C07321=1192.397,329.758,-73.014,-176.371,7.845,148.458
C07322=1192.393,330.005,-73.045,-176.368,7.848,148.458
C07323=1192.389,330.253,-73.077,-176.366,7.851,148.458
C07324=1192.384,330.501,-73.109,-176.363,7.855,148.459
C07325=1192.381,330.749,-73.141,-176.361,7.858,148.459
C07326=1192.377,330.997,-73.173,-176.359,7.860,148.459
C07327=1192.372,331.245,-73.205,-176.357,7.864,148.459
C07328=1192.368,331.493,-73.237,-176.354,7.867,148.459
C07329=1192.364,331.741,-73.268,-176.352,7.870,148.459
C07330=1192.359,331.989,-73.300,-176.350,7.873,148.459
C07331=1192.355,332.237,-73.332,-176.347,7.875,148.459
C07332=1192.352,332.485,-73.363,-176.345,7.879,148.460
C07333=1192.347,332.733,-73.395,-176.342,7.882,148.460
C07334=1192.343,332.981,-73.427,-176.340,7.885,148.460
C07335=1192.339,333.229,-73.459,-176.338,7.888,148.460
C07336=1192.334,333.476,-73.491,-176.335,7.892,148.460
C07337=1192.331,333.724,-73.524,-176.334,7.894,148.460
C07338=1192.327,333.972,-73.556,-176.331,7.897,148.460
C07339=1192.322,334.220,-73.588,-176.329,7.900,148.460
C07340=1192.318,334.468,-73.620,-176.326,7.904,148.461
C07341=1192.314,334.716,-73.652,-176.324,7.907,148.461
C07342=1192.310,334.963,-73.683,-176.321,7.910,148.461
C07343=1192.305,335.212,-73.716,-176.320,7.913,148.461
C07344=1192.301,335.460,-73.748,-176.318,7.916,148.461
C07345=1192.298,335.708,-73.780,-176.315,7.919,148.461
C07346=1192.293,335.955,-73.812,-176.313,7.922,148.461
C07347=1192.289,336.203,-73.844,-176.310,7.926,148.462
C07348=1192.285,336.451,-73.877,-176.308,7.929,148.462
C07349=1192.281,336.699,-73.909,-176.306,7.931,148.462
C07350=1192.276,336.947,-73.941,-176.304,7.934,148.462
C07351=1192.273,337.194,-73.973,-176.302,7.938,148.462
C07352=1192.268,337.443,-74.006,-176.299,7.941,148.462
C07353=1192.265,337.691,-74.037,-176.297,7.944,148.463
C07354=1192.260,337.938,-74.070,-176.294,7.947,148.463
C07355=1192.256,338.186,-74.102,-176.293,7.950,148.463
C07356=1192.252,338.434,-74.135,-176.290,7.953,148.463
C07357=1192.248,338.682,-74.166,-176.288,7.956,148.463
C07358=1192.244,338.930,-74.199,-176.286,7.960,148.463
C07359=1192.240,339.177,-74.231,-176.283,7.963,148.464
C07360=1192.235,339.425,-74.263,-176.281,7.966,148.464
C07361=1192.231,339.674,-74.296,-176.279,7.969,148.464
C07362=1192.227,339.921,-74.328,-176.277,7.972,148.464
C07363=1192.223,340.200,-74.365,-176.274,7.976,148.464
C07364=1192.218,340.479,-74.401,-176.272,7.979,148.464
C07365=1192.212,340.757,-74.438,-176.269,7.982,148.465
C07366=1192.208,341.036,-74.474,-176.267,7.987,148.465
C07367=1192.204,341.284,-74.506,-176.265,7.989,148.465
C07368=1192.200,341.531,-74.539,-176.263,7.992,148.465
C07369=1192.195,341.780,-74.572,-176.260,7.996,148.465
C07370=1192.192,342.027,-74.604,-176.258,7.999,148.466
C07371=1192.188,342.276,-74.637,-176.255,8.002,148.466
C07372=1192.183,342.523,-74.669,-176.253,8.005,148.466
C07373=1192.179,342.771,-74.701,-176.252,8.008,148.466
C07374=1192.175,343.018,-74.734,-176.249,8.011,148.466
C07375=1192.171,343.267,-74.767,-176.247,8.015,148.467
C07376=1192.167,343.514,-74.799,-176.245,8.018,148.467
C07377=1192.163,343.763,-74.832,-176.243,8.021,148.467
C07378=1192.159,344.010,-74.865,-176.240,8.025,148.467
C07379=1192.154,344.257,-74.898,-176.239,8.027,148.467
C07380=1192.150,344.505,-74.930,-176.236,8.030,148.468
C07381=1192.146,344.753,-74.963,-176.234,8.034,148.468
C07382=1192.142,345.001,-74.995,-176.232,8.037,148.468
C07383=1192.137,345.249,-75.028,-176.230,8.040,148.468
C07384=1192.134,345.497,-75.061,-176.227,8.044,148.468
C07385=1192.130,345.745,-75.093,-176.226,8.046,148.469
C07386=1192.125,345.993,-75.127,-176.224,8.050,148.469
C07387=1192.121,346.240,-75.160,-176.221,8.053,148.469
C07388=1192.118,346.488,-75.192,-176.219,8.056,148.469
C07389=1192.113,346.736,-75.225,-176.217,8.060,148.470
C07390=1192.109,346.983,-75.258,-176.215,8.063,148.470
C07391=1192.104,347.231,-75.290,-176.213,8.065,148.470
C07392=1192.100,347.479,-75.323,-176.211,8.069,148.470
C07393=1192.096,347.727,-75.356,-176.208,8.072,148.470
C07394=1192.093,347.974,-75.389,-176.206,8.075,148.471
C07395=1192.088,348.223,-75.421,-176.204,8.079,148.471
C07396=1192.084,348.470,-75.454,-176.202,8.082,148.471
C07397=1192.080,348.718,-75.488,-176.199,8.085,148.471
C07398=1192.076,348.966,-75.521,-176.198,8.088,148.471
C07399=1192.072,349.214,-75.554,-176.196,8.091,148.472
C07400=1192.067,349.461,-75.587,-176.194,8.095,148.472
C07401=1192.063,349.710,-75.620,-176.191,8.098,148.472
C07402=1192.060,349.957,-75.652,-176.189,8.101,148.473
C07403=1192.056,350.205,-75.685,-176.187,8.105,148.473
C07404=1192.051,350.453,-75.718,-176.185,8.107,148.473
C07405=1192.047,350.700,-75.752,-176.183,8.111,148.473
C07406=1192.043,350.948,-75.785,-176.181,8.114,148.474
C07407=1192.039,351.196,-75.818,-176.179,8.118,148.474
C07408=1192.035,351.444,-75.851,-176.177,8.121,148.474
C07409=1192.031,351.691,-75.884,-176.175,8.124,148.474
C07410=1192.027,351.939,-75.917,-176.173,8.127,148.474
C07411=1192.022,352.187,-75.951,-176.171,8.130,148.475
C07412=1192.018,352.434,-75.984,-176.169,8.134,148.475
C07413=1192.014,352.682,-76.017,-176.167,8.137,148.475
C07414=1192.010,352.930,-76.050,-176.164,8.140,148.476
C07415=1192.006,353.178,-76.083,-176.163,8.144,148.476
C07416=1192.002,353.425,-76.116,-176.161,8.146,148.476
C07417=1191.998,353.674,-76.150,-176.159,8.150,148.476
C07418=1191.994,353.922,-76.183,-176.156,8.153,148.477
C07419=1191.990,354.169,-76.216,-176.155,8.157,148.477
C07420=1191.986,354.417,-76.249,-176.152,8.160,148.477
C07421=1191.982,354.665,-76.282,-176.150,8.163,148.477
C07422=1191.977,354.912,-76.316,-176.149,8.166,148.478
C07423=1191.973,355.160,-76.349,-176.147,8.169,148.478
C07424=1191.969,355.408,-76.382,-176.144,8.173,148.478
C07425=1191.965,355.656,-76.415,-176.143,8.176,148.479
C07426=1191.961,355.903,-76.449,-176.140,8.180,148.479
C07427=1191.957,356.150,-76.482,-176.139,8.183,148.479
C07428=1191.953,356.399,-76.516,-176.137,8.186,148.480
C07429=1191.949,356.647,-76.549,-176.135,8.189,148.480
C07430=1191.945,356.895,-76.583,-176.133,8.193,148.480
C07431=1191.941,357.142,-76.616,-176.131,8.196,148.480
C07432=1191.937,357.389,-76.650,-176.129,8.200,148.481
C07433=1191.932,357.637,-76.683,-176.127,8.203,148.481
C07434=1191.928,357.885,-76.716,-176.125,8.206,148.481
C07435=1191.925,358.133,-76.750,-176.123,8.209,148.482
C07436=1191.920,358.381,-76.784,-176.121,8.213,148.482
C07437=1191.916,358.629,-76.817,-176.119,8.216,148.482
C07438=1191.912,358.876,-76.850,-176.117,8.220,148.483
C07439=1191.908,359.123,-76.884,-176.115,8.223,148.483
C07440=1191.904,359.371,-76.917,-176.113,8.226,148.483
C07441=1191.900,359.620,-76.951,-176.112,8.229,148.484
C07442=1191.896,359.867,-76.985,-176.110,8.233,148.484
C07443=1191.892,360.115,-77.018,-176.108,8.236,148.484
C07444=1191.888,360.362,-77.052,-176.106,8.240,148.485
C07445=1191.884,360.610,-77.085,-176.104,8.242,148.485
C07446=1191.879,360.858,-77.119,-176.102,8.246,148.485
C07447=1191.876,361.105,-77.153,-176.100,8.249,148.486
C07448=1191.871,361.353,-77.186,-176.098,8.253,148.486
C07449=1191.868,361.600,-77.220,-176.097,8.256,148.486
C07450=1191.863,361.848,-77.254,-176.095,8.259,148.487
C07451=1191.860,362.096,-77.288,-176.093,8.263,148.487
C07452=1191.855,362.344,-77.322,-176.091,8.266,148.488
C07453=1191.851,362.592,-77.355,-176.090,8.269,148.488
C07454=1191.847,362.839,-77.389,-176.088,8.273,148.488
C07455=1191.843,363.087,-77.423,-176.086,8.276,148.489
C07456=1191.839,363.334,-77.457,-176.084,8.280,148.489
C07457=1191.836,363.582,-77.490,-176.082,8.282,148.489
C07458=1191.831,363.830,-77.524,-176.081,8.286,148.490
C07459=1191.827,364.077,-77.558,-176.079,8.290,148.490
C07460=1191.823,364.325,-77.592,-176.078,8.292,148.490
C07461=1191.819,364.573,-77.626,-176.076,8.296,148.491
C07462=1191.815,364.820,-77.659,-176.074,8.299,148.491
C07463=1191.811,365.068,-77.693,-176.072,8.302,148.491
C07464=1191.807,365.316,-77.728,-176.071,8.306,148.492
C07465=1191.803,365.563,-77.761,-176.069,8.309,148.492
C07466=1191.799,365.811,-77.796,-176.068,8.312,148.493
C07467=1191.794,366.092,-77.834,-176.065,8.317,148.493
C07468=1191.789,366.373,-77.872,-176.063,8.320,148.494
C07469=1191.785,366.655,-77.911,-176.062,8.324,148.494
C07470=1191.780,366.935,-77.949,-176.060,8.328,148.495
C07471=1191.777,367.183,-77.984,-176.058,8.331,148.495
C07472=1191.772,367.431,-78.017,-176.057,8.334,148.495
C07473=1191.768,367.678,-78.051,-176.055,8.338,148.496
C07474=1191.764,367.926,-78.086,-176.054,8.340,148.496
C07475=1191.760,368.174,-78.119,-176.052,8.344,148.497
C07476=1191.756,368.421,-78.153,-176.050,8.348,148.497
C07477=1191.752,368.669,-78.188,-176.049,8.350,148.497
C07478=1191.748,368.916,-78.222,-176.047,8.354,148.498
C07479=1191.744,369.164,-78.256,-176.046,8.357,148.498
C07480=1191.740,369.412,-78.290,-176.044,8.360,148.499
C07481=1191.736,369.660,-78.324,-176.043,8.363,148.499
C07482=1191.732,369.907,-78.358,-176.041,8.367,148.500
C07483=1191.728,370.155,-78.393,-176.040,8.371,148.500
C07484=1191.724,370.402,-78.427,-176.039,8.374,148.501
C07485=1191.719,370.650,-78.461,-176.037,8.377,148.501
C07486=1191.716,370.898,-78.495,-176.035,8.380,148.501
C07487=1191.711,371.145,-78.529,-176.034,8.384,148.502
C07488=1191.707,371.392,-78.563,-176.032,8.386,148.502
C07489=1191.704,371.640,-78.598,-176.031,8.390,148.503
C07490=1191.700,371.888,-78.632,-176.030,8.393,148.503
C07491=1191.696,372.136,-78.667,-176.029,8.396,148.504
C07492=1191.692,372.383,-78.701,-176.027,8.400,148.504
C07493=1191.687,372.631,-78.734,-176.026,8.403,148.505
C07494=1191.683,372.879,-78.769,-176.024,8.406,148.505
C07495=1191.679,373.126,-78.803,-176.023,8.409,148.505
C07496=1191.675,373.374,-78.838,-176.021,8.413,148.506
C07497=1191.671,373.621,-78.872,-176.020,8.416,148.506
C07498=1191.667,373.869,-78.906,-176.019,8.420,148.507
C07499=1191.663,374.117,-78.941,-176.017,8.422,148.507
C07500=1191.659,374.364,-78.975,-176.017,8.425,148.508
C07501=1191.655,374.612,-79.010,-176.015,8.429,148.508
C07502=1191.651,374.859,-79.044,-176.014,8.432,148.509
C07503=1191.647,375.107,-79.078,-176.013,8.435,148.509
C07504=1191.643,375.355,-79.113,-176.011,8.439,148.510
C07505=1191.639,375.602,-79.147,-176.010,8.442,148.510
C07506=1191.635,375.850,-79.182,-176.009,8.444,148.511
C07507=1191.631,376.097,-79.216,-176.008,8.448,148.511
C07508=1191.627,376.345,-79.250,-176.006,8.451,148.512
C07509=1191.623,376.592,-79.286,-176.006,8.454,148.512
C07510=1191.620,376.840,-79.320,-176.004,8.458,148.513
C07511=1191.615,377.087,-79.354,-176.003,8.461,148.513
C07512=1191.610,377.335,-79.389,-176.002,8.464,148.514
C07513=1191.606,377.583,-79.424,-176.001,8.467,148.514
C07514=1191.603,377.830,-79.457,-175.999,8.471,148.515
C07515=1191.599,378.078,-79.492,-175.998,8.474,148.515
C07516=1191.594,378.325,-79.527,-175.997,8.476,148.516
C07517=1191.591,378.573,-79.562,-175.996,8.480,148.516
C07518=1191.587,378.820,-79.596,-175.995,8.484,148.517
C07519=1191.583,379.068,-79.631,-175.994,8.486,148.517
C07520=1191.579,379.315,-79.665,-175.993,8.489,148.518
C07521=1191.575,379.563,-79.700,-175.992,8.492,148.518
C07522=1191.570,379.811,-79.734,-175.991,8.495,148.519
C07523=1191.567,380.058,-79.770,-175.990,8.498,148.519
C07524=1191.563,380.305,-79.804,-175.988,8.502,148.520
C07525=1191.559,380.553,-79.838,-175.987,8.505,148.520
C07526=1191.554,380.801,-79.873,-175.987,8.508,148.521
C07527=1191.551,381.048,-79.908,-175.985,8.511,148.521
C07528=1191.547,381.295,-79.942,-175.985,8.514,148.522
C07529=1191.543,381.544,-79.977,-175.984,8.517,148.523
C07530=1191.538,381.791,-80.012,-175.983,8.520,148.523
C07531=1191.535,382.039,-80.047,-175.982,8.523,148.524
C07532=1191.530,382.286,-80.082,-175.981,8.526,148.524
C07533=1191.527,382.534,-80.116,-175.980,8.529,148.525
C07534=1191.522,382.781,-80.150,-175.979,8.532,148.525
C07535=1191.519,383.029,-80.186,-175.979,8.536,148.526
C07536=1191.514,383.276,-80.220,-175.977,8.538,148.526
C07537=1191.510,383.524,-80.255,-175.977,8.541,148.527
C07538=1191.506,383.771,-80.290,-175.976,8.545,148.527
C07539=1191.502,384.019,-80.325,-175.975,8.548,148.528
C07540=1191.499,384.267,-80.359,-175.974,8.551,148.529
C07541=1191.494,384.514,-80.395,-175.973,8.554,148.529
C07542=1191.490,384.762,-80.429,-175.973,8.557,148.530
C07543=1191.486,385.009,-80.465,-175.972,8.560,148.530
C07544=1191.483,385.256,-80.499,-175.971,8.563,148.531
C07545=1191.478,385.504,-80.533,-175.970,8.566,148.531
C07546=1191.475,385.751,-80.569,-175.970,8.568,148.532
C07547=1191.470,385.999,-80.603,-175.969,8.571,148.533
C07548=1191.466,386.246,-80.639,-175.968,8.574,148.533
C07549=1191.462,386.494,-80.674,-175.967,8.577,148.534
C07550=1191.458,386.742,-80.708,-175.966,8.581,148.534
C07551=1191.454,386.989,-80.744,-175.966,8.583,148.535
C07552=1191.450,387.236,-80.778,-175.965,8.586,148.535
C07553=1191.447,387.484,-80.813,-175.965,8.589,148.536
C07554=1191.443,387.732,-80.848,-175.964,8.592,148.537
C07555=1191.438,387.979,-80.883,-175.964,8.594,148.537
C07556=1191.434,388.227,-80.918,-175.963,8.598,148.538
C07557=1191.430,388.474,-80.953,-175.962,8.601,148.538
C07558=1191.426,388.722,-80.988,-175.961,8.604,148.539
C07559=1191.423,388.969,-81.024,-175.961,8.606,148.539
C07560=1191.418,389.217,-81.058,-175.960,8.609,148.540
C07561=1191.414,389.464,-81.094,-175.960,8.611,148.540
C07562=1191.410,389.712,-81.128,-175.959,8.614,148.541
C07563=1191.407,389.959,-81.163,-175.959,8.618,148.542
C07564=1191.403,390.207,-81.198,-175.958,8.620,148.542
C07565=1191.399,390.454,-81.233,-175.958,8.623,148.543
C07566=1191.395,390.702,-81.268,-175.957,8.626,148.544
C07567=1191.390,390.949,-81.303,-175.957,8.629,148.544
C07568=1191.386,391.197,-81.338,-175.956,8.632,148.545
C07569=1191.383,391.444,-81.373,-175.956,8.634,148.545
C07570=1191.378,391.692,-81.408,-175.955,8.637,148.546
C07571=1191.374,391.975,-81.449,-175.954,8.640,148.547
C07572=1191.369,392.259,-81.489,-175.954,8.643,148.547
C07573=1191.365,392.542,-81.529,-175.954,8.646,148.548
C07574=1191.360,392.825,-81.569,-175.953,8.649,148.548
C07575=1191.356,393.073,-81.604,-175.952,8.652,148.549
C07576=1191.353,393.321,-81.640,-175.952,8.655,148.550
C07577=1191.348,393.568,-81.674,-175.952,8.657,148.550
C07578=1191.344,393.815,-81.710,-175.951,8.660,148.551
C07579=1191.340,394.062,-81.745,-175.951,8.662,148.551
C07580=1191.336,394.310,-81.780,-175.950,8.666,148.552
C07581=1191.333,394.558,-81.815,-175.950,8.668,148.553
C07582=1191.328,394.805,-81.850,-175.950,8.670,148.553
C07583=1191.324,395.053,-81.885,-175.949,8.673,148.554
C07584=1191.321,395.300,-81.921,-175.949,8.676,148.554
C07585=1191.316,395.547,-81.956,-175.948,8.679,148.555
C07586=1191.312,395.795,-81.991,-175.948,8.681,148.555
C07587=1191.309,396.043,-82.026,-175.948,8.683,148.556
C07588=1191.304,396.290,-82.062,-175.947,8.687,148.557
C07589=1191.301,396.538,-82.096,-175.947,8.689,148.557
C07590=1191.297,396.785,-82.132,-175.947,8.691,148.558
C07591=1191.293,397.032,-82.167,-175.947,8.694,148.558
C07592=1191.289,397.280,-82.202,-175.946,8.697,148.559
C07593=1191.284,397.528,-82.238,-175.946,8.699,148.560
C07594=1191.280,397.775,-82.273,-175.946,8.701,148.560
C07595=1191.276,398.022,-82.309,-175.945,8.704,148.561
C07596=1191.272,398.270,-82.344,-175.945,8.707,148.561
C07597=1191.269,398.518,-82.379,-175.945,8.709,148.562
C07598=1191.264,398.765,-82.414,-175.944,8.711,148.562
C07599=1191.260,399.013,-82.449,-175.944,8.714,148.563
C07600=1191.257,399.260,-82.485,-175.944,8.716,148.563
C07601=1191.253,399.507,-82.520,-175.944,8.719,148.564
C07602=1191.249,399.755,-82.556,-175.943,8.722,148.565
C07603=1191.245,400.002,-82.591,-175.943,8.724,148.565
C07604=1191.241,400.249,-82.626,-175.943,8.726,148.566
C07605=1191.237,400.497,-82.661,-175.943,8.728,148.566
C07606=1191.233,400.745,-82.697,-175.943,8.731,148.567
C07607=1191.228,400.992,-82.732,-175.943,8.733,148.568
C07608=1191.224,401.240,-82.767,-175.942,8.736,148.568
C07609=1191.221,401.487,-82.803,-175.942,8.739,148.569
C07610=1191.217,401.735,-82.838,-175.941,8.741,148.569
C07611=1191.213,401.981,-82.874,-175.941,8.743,148.570
C07612=1191.209,402.229,-82.909,-175.941,8.746,148.570
C07613=1191.205,402.477,-82.944,-175.941,8.748,148.571
C07614=1191.201,402.724,-82.979,-175.941,8.750,148.572
C07615=1191.196,402.972,-83.015,-175.941,8.753,148.572
C07616=1191.193,403.219,-83.051,-175.940,8.755,148.573
C07617=1191.189,403.467,-83.086,-175.940,8.757,148.573
C07618=1191.185,403.714,-83.121,-175.940,8.760,148.574
C07619=1191.181,403.962,-83.156,-175.940,8.762,148.574
C07620=1191.177,404.209,-83.192,-175.940,8.764,148.575
C07621=1191.174,404.457,-83.227,-175.939,8.766,148.575
C07622=1191.169,404.704,-83.263,-175.939,8.769,148.576
C07623=1191.165,404.951,-83.299,-175.939,8.771,148.576
C07624=1191.161,405.199,-83.334,-175.939,8.773,148.577
C07625=1191.157,405.446,-83.369,-175.939,8.776,148.578
C07626=1191.153,405.693,-83.405,-175.939,8.778,148.578
C07627=1191.149,405.941,-83.440,-175.938,8.780,148.579
C07628=1191.146,406.189,-83.475,-175.938,8.783,148.579
C07629=1191.141,406.436,-83.511,-175.938,8.785,148.580
C07630=1191.137,406.683,-83.547,-175.938,8.787,148.580
C07631=1191.133,406.931,-83.582,-175.937,8.789,148.581
C07632=1191.130,407.178,-83.618,-175.938,8.792,148.582
C07633=1191.125,407.425,-83.653,-175.938,8.793,148.582
C07634=1191.121,407.673,-83.689,-175.938,8.796,148.583
C07635=1191.117,407.920,-83.725,-175.937,8.798,148.583
C07636=1191.114,408.168,-83.760,-175.937,8.800,148.584
C07637=1191.110,408.415,-83.796,-175.937,8.802,148.584
C07638=1191.105,408.663,-83.830,-175.937,8.805,148.585
C07639=1191.102,408.910,-83.866,-175.936,8.807,148.585
C07640=1191.097,409.158,-83.902,-175.936,8.809,148.586
C07641=1191.094,409.406,-83.937,-175.937,8.811,148.586
C07642=1191.089,409.652,-83.973,-175.937,8.813,148.587
C07643=1191.086,409.900,-84.008,-175.936,8.816,148.587
C07644=1191.082,410.147,-84.044,-175.936,8.818,148.588
C07645=1191.078,410.395,-84.080,-175.936,8.820,148.588
C07646=1191.073,410.642,-84.115,-175.936,8.822,148.589
C07647=1191.070,410.890,-84.151,-175.936,8.824,148.589
C07648=1191.066,411.137,-84.186,-175.936,8.826,148.590
C07649=1191.062,411.385,-84.222,-175.936,8.828,148.591
C07650=1191.058,411.632,-84.258,-175.935,8.831,148.591
C07651=1191.054,411.879,-84.293,-175.935,8.833,148.592
C07652=1191.050,412.127,-84.329,-175.935,8.834,148.592
C07653=1191.046,412.374,-84.364,-175.935,8.837,148.593
C07654=1191.042,412.622,-84.400,-175.935,8.839,148.593
C07655=1191.038,412.869,-84.435,-175.935,8.841,148.594
C07656=1191.034,413.116,-84.471,-175.935,8.842,148.594
C07657=1191.031,413.364,-84.507,-175.935,8.845,148.595
C07658=1191.026,413.612,-84.543,-175.934,8.847,148.595
C07659=1191.022,413.859,-84.578,-175.934,8.849,148.596
C07660=1191.018,414.106,-84.613,-175.934,8.851,148.596
C07661=1191.015,414.353,-84.649,-175.934,8.853,148.597
C07662=1191.010,414.601,-84.685,-175.934,8.855,148.597
C07663=1191.006,414.849,-84.721,-175.934,8.857,148.598
C07664=1191.003,415.096,-84.756,-175.934,8.859,148.598
C07665=1190.999,415.343,-84.791,-175.934,8.861,148.599
C07666=1190.994,415.591,-84.828,-175.934,8.863,148.599
C07667=1190.988,415.973,-84.883,-175.934,8.866,148.600
C07668=1190.984,416.354,-84.938,-175.933,8.869,148.601
C07669=1190.984,416.736,-84.992,-175.934,8.872,148.601
C07670=1190.987,417.117,-85.046,-175.933,8.875,148.602
C07671=1190.566,417.117,-85.087,-175.936,8.886,148.606
C07672=1190.562,416.734,-85.032,-175.937,8.883,148.605
C07673=1190.564,416.349,-84.978,-175.936,8.880,148.604
C07674=1190.567,415.965,-84.922,-175.937,8.877,148.604
C07675=1190.573,415.580,-84.866,-175.937,8.874,148.603
C07676=1190.577,415.332,-84.830,-175.937,8.872,148.602
C07677=1190.581,415.085,-84.795,-175.937,8.870,148.602
C07678=1190.585,414.838,-84.759,-175.937,8.868,148.601
C07679=1190.589,414.590,-84.724,-175.937,8.866,148.601
C07680=1190.593,414.342,-84.688,-175.937,8.864,148.600
C07681=1190.597,414.095,-84.652,-175.938,8.861,148.600
C07682=1190.601,413.848,-84.617,-175.937,8.860,148.599
C07683=1190.605,413.601,-84.581,-175.938,8.858,148.599
C07684=1190.609,413.353,-84.545,-175.938,8.855,148.598
C07685=1190.613,413.105,-84.510,-175.937,8.854,148.598
C07686=1190.617,412.858,-84.474,-175.938,8.852,148.597
C07687=1190.621,412.611,-84.439,-175.938,8.849,148.597
C07688=1190.625,412.363,-84.403,-175.938,8.847,148.596
C07689=1190.629,412.116,-84.367,-175.938,8.845,148.596
C07690=1190.633,411.868,-84.332,-175.938,8.843,148.595
C07691=1190.636,411.621,-84.296,-175.938,8.841,148.595
C07692=1190.641,411.374,-84.260,-175.939,8.839,148.594
C07693=1190.645,411.126,-84.225,-175.939,8.837,148.594
C07694=1190.649,410.879,-84.189,-175.939,8.835,148.593
C07695=1190.652,410.631,-84.154,-175.939,8.833,148.593
C07696=1190.656,410.384,-84.118,-175.939,8.831,148.592
C07697=1190.661,410.136,-84.083,-175.939,8.828,148.592
C07698=1190.665,409.889,-84.047,-175.940,8.826,148.591
C07699=1190.668,409.641,-84.011,-175.939,8.824,148.590
C07700=1190.672,409.394,-83.976,-175.939,8.822,148.590
C07701=1190.676,409.147,-83.941,-175.939,8.820,148.589
C07702=1190.680,408.899,-83.905,-175.940,8.818,148.589
C07703=1190.684,408.652,-83.869,-175.940,8.815,148.588
C07704=1190.688,408.404,-83.833,-175.940,8.813,148.588
C07705=1190.692,408.158,-83.798,-175.940,8.811,148.587
C07706=1190.696,407.910,-83.763,-175.940,8.809,148.587
C07707=1190.700,407.662,-83.727,-175.940,8.807,148.586
C07708=1190.704,407.415,-83.691,-175.940,8.805,148.586
C07709=1190.708,407.167,-83.657,-175.940,8.802,148.585
C07710=1190.712,406.920,-83.621,-175.941,8.800,148.585
C07711=1190.716,406.672,-83.585,-175.941,8.798,148.584
C07712=1190.719,406.425,-83.550,-175.941,8.796,148.583
C07713=1190.724,406.177,-83.514,-175.941,8.793,148.583
C07714=1190.728,405.930,-83.479,-175.942,8.791,148.582
C07715=1190.732,405.683,-83.443,-175.941,8.788,148.582
C07716=1190.735,405.435,-83.408,-175.942,8.786,148.581
C07717=1190.739,405.188,-83.372,-175.942,8.784,148.581
C07718=1190.743,404.941,-83.337,-175.942,8.782,148.580
C07719=1190.748,404.692,-83.301,-175.942,8.779,148.580
C07720=1190.752,404.445,-83.266,-175.943,8.777,148.579
C07721=1190.756,404.198,-83.231,-175.942,8.776,148.579
C07722=1190.760,403.951,-83.195,-175.942,8.773,148.578
C07723=1190.763,403.703,-83.160,-175.943,8.770,148.577
C07724=1190.767,403.456,-83.124,-175.943,8.768,148.577
C07725=1190.772,403.209,-83.088,-175.943,8.765,148.576
C07726=1190.776,402.960,-83.053,-175.944,8.763,148.576
C07727=1190.780,402.713,-83.018,-175.943,8.761,148.575
C07728=1190.783,402.465,-82.982,-175.944,8.758,148.574
C07729=1190.787,402.219,-82.947,-175.944,8.756,148.574
C07730=1190.791,401.971,-82.912,-175.944,8.754,148.573
C07731=1190.795,401.724,-82.876,-175.944,8.752,148.573
C07732=1190.799,401.476,-82.842,-175.945,8.749,148.572
C07733=1190.804,401.228,-82.805,-175.944,8.747,148.572
C07734=1190.807,400.981,-82.770,-175.945,8.744,148.571
C07735=1190.811,400.733,-82.734,-175.945,8.742,148.571
C07736=1190.815,400.487,-82.699,-175.945,8.740,148.570
C07737=1190.819,400.238,-82.664,-175.946,8.737,148.569
C07738=1190.823,399.991,-82.629,-175.946,8.734,148.569
C07739=1190.827,399.744,-82.594,-175.946,8.732,148.568
C07740=1190.831,399.497,-82.558,-175.946,8.730,148.568
C07741=1190.835,399.249,-82.522,-175.947,8.727,148.567
C07742=1190.839,399.002,-82.488,-175.947,8.725,148.567
C07743=1190.843,398.754,-82.452,-175.947,8.722,148.566
C07744=1190.847,398.506,-82.416,-175.947,8.720,148.565
C07745=1190.851,398.259,-82.381,-175.948,8.717,148.565
C07746=1190.855,398.012,-82.346,-175.948,8.715,148.564
C07747=1190.859,397.764,-82.311,-175.948,8.713,148.564
C07748=1190.863,397.517,-82.275,-175.949,8.709,148.563
C07749=1190.867,397.269,-82.241,-175.949,8.707,148.562
C07750=1190.871,397.022,-82.205,-175.949,8.705,148.562
C07751=1190.875,396.774,-82.170,-175.949,8.703,148.561
C07752=1190.879,396.527,-82.134,-175.950,8.699,148.561
C07753=1190.883,396.279,-82.100,-175.950,8.697,148.560
C07754=1190.887,396.032,-82.064,-175.950,8.695,148.560
C07755=1190.891,395.785,-82.029,-175.951,8.692,148.559
C07756=1190.895,395.537,-81.994,-175.951,8.689,148.558
C07757=1190.898,395.289,-81.959,-175.951,8.687,148.558
C07758=1190.903,395.042,-81.923,-175.952,8.684,148.557
C07759=1190.907,394.794,-81.888,-175.952,8.681,148.557
C07760=1190.910,394.547,-81.853,-175.952,8.679,148.556
C07761=1190.915,394.300,-81.818,-175.953,8.676,148.555
C07762=1190.919,394.052,-81.783,-175.953,8.674,148.555
C07763=1190.922,393.804,-81.747,-175.954,8.671,148.554
C07764=1190.927,393.558,-81.712,-175.954,8.668,148.554
C07765=1190.930,393.310,-81.677,-175.954,8.666,148.553
C07766=1190.934,393.062,-81.642,-175.955,8.663,148.553
C07767=1190.938,392.815,-81.607,-175.955,8.660,148.552
C07768=1190.943,392.531,-81.567,-175.956,8.657,148.551
C07769=1190.948,392.248,-81.526,-175.956,8.654,148.551
C07770=1190.952,391.964,-81.486,-175.957,8.651,148.550
C07771=1190.957,391.681,-81.445,-175.957,8.647,148.549
C07772=1190.961,391.433,-81.410,-175.958,8.645,148.549
C07773=1190.964,391.186,-81.376,-175.959,8.642,148.548
C07774=1190.969,390.938,-81.341,-175.959,8.640,148.548
C07775=1190.972,390.691,-81.306,-175.960,8.637,148.547
C07776=1190.977,390.444,-81.271,-175.960,8.634,148.547
C07777=1190.981,390.196,-81.235,-175.961,8.631,148.546
C07778=1190.984,389.949,-81.200,-175.961,8.628,148.545
C07779=1190.989,389.701,-81.165,-175.961,8.626,148.545
C07780=1190.993,389.454,-81.130,-175.962,8.623,148.544
C07781=1190.997,389.205,-81.095,-175.963,8.619,148.543
C07782=1191.001,388.959,-81.060,-175.963,8.617,148.543
C07783=1191.005,388.711,-81.025,-175.964,8.614,148.542
C07784=1191.009,388.464,-80.990,-175.965,8.611,148.542
C07785=1191.013,388.216,-80.955,-175.965,8.609,148.541
C07786=1191.017,387.968,-80.920,-175.966,8.606,148.541
C07787=1191.021,387.721,-80.885,-175.966,8.603,148.540
C07788=1191.024,387.474,-80.850,-175.967,8.600,148.540
C07789=1191.029,387.226,-80.816,-175.968,8.597,148.539
C07790=1191.033,386.978,-80.781,-175.968,8.594,148.538
C07791=1191.037,386.731,-80.746,-175.969,8.591,148.538
C07792=1191.041,386.483,-80.711,-175.970,8.588,148.537
C07793=1191.045,386.236,-80.675,-175.970,8.586,148.537
C07794=1191.049,385.988,-80.641,-175.971,8.582,148.536
C07795=1191.053,385.741,-80.605,-175.972,8.579,148.535
C07796=1191.057,385.494,-80.571,-175.973,8.576,148.535
C07797=1191.061,385.245,-80.537,-175.973,8.573,148.534
C07798=1191.064,384.998,-80.501,-175.974,8.570,148.534
C07799=1191.069,384.751,-80.467,-175.975,8.567,148.533
C07800=1191.072,384.503,-80.431,-175.975,8.565,148.533
C07801=1191.077,384.256,-80.396,-175.976,8.562,148.532
C07802=1191.081,384.007,-80.362,-175.977,8.559,148.532
C07803=1191.085,383.761,-80.327,-175.978,8.556,148.531
C07804=1191.089,383.513,-80.292,-175.979,8.553,148.530
C07805=1191.093,383.265,-80.258,-175.980,8.550,148.530
C07806=1191.097,383.018,-80.222,-175.980,8.546,148.529
C07807=1191.101,382.771,-80.188,-175.981,8.543,148.529
C07808=1191.105,382.523,-80.154,-175.982,8.541,148.528
C07809=1191.108,382.275,-80.118,-175.983,8.537,148.528
C07810=1191.113,382.028,-80.084,-175.984,8.534,148.527
C07811=1191.117,381.780,-80.049,-175.985,8.531,148.527
C07812=1191.121,381.533,-80.014,-175.986,8.528,148.526
C07813=1191.124,381.285,-79.979,-175.987,8.525,148.526
C07814=1191.129,381.038,-79.945,-175.988,8.521,148.525
C07815=1191.133,380.790,-79.910,-175.989,8.518,148.524
C07816=1191.137,380.543,-79.875,-175.990,8.515,148.524
C07817=1191.141,380.295,-79.840,-175.991,8.512,148.523
C07818=1191.145,380.047,-79.806,-175.992,8.509,148.523
C07819=1191.149,379.799,-79.771,-175.993,8.506,148.522
C07820=1191.153,379.552,-79.737,-175.994,8.503,148.522
C07821=1191.157,379.304,-79.701,-175.995,8.499,148.521
C07822=1191.161,379.057,-79.667,-175.996,8.496,148.521
C07823=1191.165,378.809,-79.633,-175.997,8.494,148.520
C07824=1191.169,378.562,-79.598,-175.998,8.490,148.520
C07825=1191.173,378.314,-79.564,-175.999,8.488,148.519
C07826=1191.177,378.067,-79.529,-176.001,8.484,148.519
C07827=1191.181,377.819,-79.494,-176.002,8.481,148.518
C07828=1191.185,377.572,-79.459,-176.003,8.478,148.518
C07829=1191.189,377.325,-79.425,-176.003,8.475,148.517
C07830=1191.193,377.076,-79.391,-176.005,8.471,148.517
C07831=1191.198,376.829,-79.356,-176.006,8.468,148.516
C07832=1191.201,376.581,-79.322,-176.007,8.465,148.516
C07833=1191.206,376.334,-79.287,-176.009,8.461,148.515
C07834=1191.210,376.086,-79.253,-176.010,8.459,148.515
C07835=1191.213,375.839,-79.218,-176.011,8.455,148.514
C07836=1191.217,375.591,-79.183,-176.013,8.452,148.514
C07837=1191.222,375.344,-79.149,-176.014,8.449,148.513
C07838=1191.226,375.097,-79.115,-176.015,8.446,148.513
C07839=1191.229,374.848,-79.080,-176.016,8.442,148.512
C07840=1191.233,374.601,-79.046,-176.017,8.439,148.512
C07841=1191.237,374.353,-79.011,-176.018,8.436,148.511
C07842=1191.242,374.106,-78.977,-176.020,8.433,148.511
C07843=1191.245,373.858,-78.943,-176.021,8.430,148.510
C07844=1191.250,373.611,-78.908,-176.023,8.426,148.510
C07845=1191.253,373.363,-78.874,-176.024,8.423,148.509
C07846=1191.257,373.115,-78.839,-176.025,8.420,148.509
C07847=1191.262,372.868,-78.805,-176.027,8.416,148.508
C07848=1191.265,372.620,-78.771,-176.028,8.414,148.508
C07849=1191.270,372.373,-78.736,-176.029,8.410,148.507
C07850=1191.274,372.125,-78.703,-176.030,8.407,148.507
C07851=1191.278,371.877,-78.668,-176.032,8.403,148.506
C07852=1191.282,371.630,-78.634,-176.033,8.401,148.506
C07853=1191.286,371.382,-78.600,-176.035,8.397,148.506
C07854=1191.290,371.134,-78.566,-176.036,8.394,148.505
C07855=1191.294,370.887,-78.531,-176.038,8.390,148.505
C07856=1191.297,370.639,-78.497,-176.039,8.387,148.504
C07857=1191.302,370.392,-78.463,-176.041,8.384,148.504
C07858=1191.307,370.144,-78.429,-176.042,8.381,148.503
C07859=1191.310,369.896,-78.395,-176.044,8.377,148.503
C07860=1191.315,369.649,-78.360,-176.045,8.374,148.502
C07861=1191.318,369.401,-78.326,-176.046,8.371,148.502
C07862=1191.322,369.153,-78.291,-176.048,8.368,148.502
C07863=1191.327,368.906,-78.258,-176.050,8.364,148.501
C07864=1191.330,368.658,-78.224,-176.051,8.361,148.501
C07865=1191.334,368.410,-78.190,-176.053,8.358,148.500
C07866=1191.338,368.163,-78.156,-176.054,8.354,148.500
C07867=1191.342,367.915,-78.121,-176.056,8.351,148.500
C07868=1191.346,367.667,-78.088,-176.057,8.348,148.499
C07869=1191.351,367.420,-78.053,-176.059,8.344,148.499
C07870=1191.355,367.173,-78.019,-176.060,8.341,148.498
C07871=1191.359,366.924,-77.985,-176.062,8.338,148.498
C07872=1191.364,366.643,-77.947,-176.064,8.334,148.497
C07873=1191.368,366.362,-77.908,-176.066,8.330,148.497
C07874=1191.373,366.082,-77.869,-176.068,8.327,148.497
C07875=1191.377,365.800,-77.831,-176.069,8.323,148.496
C07876=1191.381,365.553,-77.797,-176.071,8.319,148.496
C07877=1191.385,365.305,-77.763,-176.073,8.316,148.495
C07878=1191.389,365.057,-77.729,-176.075,8.312,148.495
C07879=1191.393,364.810,-77.696,-176.076,8.309,148.494
C07880=1191.397,364.562,-77.661,-176.078,8.306,148.494
C07881=1191.401,364.314,-77.628,-176.080,8.302,148.494
C07882=1191.405,364.067,-77.594,-176.081,8.300,148.493
C07883=1191.410,363.819,-77.560,-176.083,8.296,148.493
C07884=1191.413,363.571,-77.526,-176.085,8.292,148.492
C07885=1191.418,363.324,-77.493,-176.087,8.290,148.492
C07886=1191.422,363.076,-77.458,-176.088,8.286,148.492
C07887=1191.425,362.828,-77.424,-176.090,8.283,148.491
C07888=1191.430,362.581,-77.391,-176.092,8.279,148.491
C07889=1191.433,362.334,-77.357,-176.094,8.276,148.491
C07890=1191.438,362.085,-77.323,-176.095,8.273,148.490
C07891=1191.442,361.837,-77.290,-176.097,8.269,148.490
C07892=1191.446,361.590,-77.256,-176.099,8.266,148.490
C07893=1191.450,361.342,-77.222,-176.101,8.263,148.489
C07894=1191.454,361.094,-77.188,-176.102,8.259,148.489
C07895=1191.458,360.846,-77.155,-176.105,8.256,148.489
C07896=1191.462,360.599,-77.121,-176.107,8.253,148.488
C07897=1191.466,360.352,-77.088,-176.109,8.249,148.488
C07898=1191.471,360.104,-77.054,-176.110,8.246,148.488
C07899=1191.474,359.856,-77.020,-176.112,8.243,148.487
C07900=1191.478,359.608,-76.987,-176.114,8.239,148.487
C07901=1191.482,359.361,-76.953,-176.116,8.236,148.487
C07902=1191.486,359.113,-76.920,-176.118,8.232,148.486
C07903=1191.491,358.865,-76.886,-176.119,8.230,148.486
C07904=1191.495,358.617,-76.853,-176.122,8.226,148.486
C07905=1191.498,358.370,-76.819,-176.123,8.223,148.485
C07906=1191.502,358.122,-76.785,-176.126,8.219,148.485
C07907=1191.507,357.874,-76.752,-176.127,8.216,148.485
C07908=1191.510,357.627,-76.718,-176.130,8.212,148.484
C07909=1191.515,357.379,-76.685,-176.131,8.210,148.484
C07910=1191.519,357.131,-76.651,-176.133,8.206,148.484
C07911=1191.524,356.884,-76.618,-176.135,8.203,148.484
C07912=1191.527,356.636,-76.584,-176.137,8.199,148.483
C07913=1191.531,356.388,-76.551,-176.139,8.196,148.483
C07914=1191.535,356.140,-76.518,-176.141,8.192,148.482
C07915=1191.539,355.893,-76.485,-176.143,8.189,148.482
C07916=1191.543,355.645,-76.451,-176.145,8.187,148.482
C07917=1191.547,355.397,-76.418,-176.147,8.183,148.482
C07918=1191.552,355.150,-76.384,-176.149,8.180,148.481
C07919=1191.556,354.902,-76.351,-176.151,8.176,148.481
C07920=1191.560,354.654,-76.317,-176.153,8.173,148.481
C07921=1191.564,354.406,-76.284,-176.155,8.169,148.480
C07922=1191.568,354.158,-76.251,-176.157,8.167,148.480
C07923=1191.572,353.910,-76.218,-176.159,8.163,148.480
C07924=1191.576,353.663,-76.184,-176.161,8.160,148.480
C07925=1191.580,353.415,-76.151,-176.163,8.157,148.479
C07926=1191.585,353.167,-76.118,-176.166,8.153,148.479
C07927=1191.589,352.919,-76.085,-176.167,8.150,148.479
C07928=1191.593,352.672,-76.052,-176.170,8.146,148.479
C07929=1191.597,352.424,-76.019,-176.171,8.144,148.478
C07930=1191.601,352.176,-75.986,-176.174,8.140,148.478
C07931=1191.605,351.929,-75.952,-176.175,8.137,148.478
C07932=1191.609,351.681,-75.919,-176.178,8.133,148.478
C07933=1191.613,351.433,-75.886,-176.180,8.130,148.477
C07934=1191.618,351.185,-75.853,-176.182,8.127,148.477
C07935=1191.622,350.938,-75.820,-176.184,8.124,148.477
C07936=1191.626,350.690,-75.787,-176.186,8.121,148.476
C07937=1191.630,350.442,-75.753,-176.188,8.117,148.476
C07938=1191.633,350.195,-75.721,-176.190,8.114,148.476
C07939=1191.638,349.947,-75.688,-176.192,8.111,148.476
C07940=1191.642,349.699,-75.655,-176.194,8.107,148.476
C07941=1191.646,349.452,-75.621,-176.197,8.104,148.475
C07942=1191.650,349.203,-75.589,-176.198,8.102,148.475
C07943=1191.654,348.955,-75.556,-176.200,8.098,148.475
C07944=1191.659,348.708,-75.523,-176.202,8.095,148.475
C07945=1191.663,348.460,-75.490,-176.205,8.091,148.474
C07946=1191.667,348.212,-75.456,-176.207,8.088,148.474
C07947=1191.671,347.964,-75.425,-176.209,8.085,148.474
C07948=1191.675,347.717,-75.391,-176.211,8.082,148.474
C07949=1191.679,347.469,-75.358,-176.213,8.079,148.473
C07950=1191.683,347.221,-75.325,-176.215,8.075,148.473
C07951=1191.687,346.973,-75.293,-176.218,8.072,148.473
C07952=1191.692,346.725,-75.259,-176.220,8.069,148.473
C07953=1191.695,346.478,-75.227,-176.222,8.066,148.473
C07954=1191.699,346.230,-75.194,-176.224,8.062,148.472
C07955=1191.704,345.981,-75.161,-176.226,8.060,148.472
C07956=1191.708,345.734,-75.128,-176.228,8.056,148.472
C07957=1191.712,345.486,-75.095,-176.230,8.053,148.472
C07958=1191.716,345.238,-75.063,-176.233,8.050,148.472
C07959=1191.720,344.991,-75.030,-176.235,8.046,148.471
C07960=1191.724,344.743,-74.997,-176.237,8.043,148.471
C07961=1191.729,344.495,-74.965,-176.239,8.041,148.471
C07962=1191.732,344.247,-74.932,-176.241,8.037,148.471
C07963=1191.737,343.999,-74.900,-176.243,8.034,148.470
C07964=1191.741,343.751,-74.867,-176.246,8.031,148.470
C07965=1191.745,343.503,-74.834,-176.248,8.027,148.470
C07966=1191.749,343.256,-74.802,-176.250,8.024,148.470
C07967=1191.753,343.009,-74.769,-176.252,8.021,148.470
C07968=1191.758,342.760,-74.736,-176.254,8.018,148.469
C07969=1191.761,342.513,-74.704,-176.256,8.015,148.469
C07970=1191.766,342.264,-74.671,-176.258,8.011,148.469
C07971=1191.770,342.017,-74.638,-176.261,8.008,148.469
C07972=1191.774,341.769,-74.606,-176.263,8.005,148.469
C07973=1191.778,341.520,-74.574,-176.266,8.002,148.469
C07974=1191.783,341.273,-74.541,-176.267,7.999,148.468
C07975=1191.786,341.025,-74.509,-176.270,7.996,148.468
C07976=1191.792,340.746,-74.472,-176.272,7.992,148.468
C07977=1191.796,340.468,-74.436,-176.275,7.988,148.468
C07978=1191.801,340.189,-74.399,-176.277,7.985,148.468
C07979=1191.805,339.911,-74.362,-176.280,7.981,148.467
C07980=1191.809,339.663,-74.331,-176.282,7.979,148.467
C07981=1191.814,339.415,-74.299,-176.284,7.975,148.467
C07982=1191.818,339.167,-74.265,-176.286,7.972,148.467
C07983=1191.822,338.919,-74.234,-176.289,7.969,148.467
C07984=1191.826,338.671,-74.201,-176.291,7.966,148.467
C07985=1191.829,338.424,-74.169,-176.293,7.962,148.466
C07986=1191.834,338.176,-74.136,-176.295,7.960,148.466
C07987=1191.838,337.928,-74.105,-176.297,7.957,148.466
C07988=1191.843,337.679,-74.072,-176.300,7.954,148.466
C07989=1191.846,337.432,-74.040,-176.302,7.950,148.466
C07990=1191.850,337.184,-74.007,-176.305,7.947,148.466
C07991=1191.855,336.936,-73.976,-176.307,7.944,148.465
C07992=1191.859,336.688,-73.943,-176.309,7.941,148.465
C07993=1191.863,336.441,-73.911,-176.311,7.938,148.465
C07994=1191.867,336.192,-73.878,-176.313,7.935,148.465
C07995=1191.871,335.945,-73.847,-176.316,7.932,148.465
C07996=1191.876,335.697,-73.814,-176.318,7.928,148.465
C07997=1191.880,335.449,-73.782,-176.321,7.925,148.464
C07998=1191.884,335.200,-73.750,-176.323,7.922,148.464
C07999=1191.888,334.953,-73.718,-176.325,7.919,148.464
C08000=1191.892,334.705,-73.686,-176.327,7.916,148.464
C08001=1191.896,334.457,-73.654,-176.329,7.913,148.464
C08002=1191.900,334.210,-73.622,-176.332,7.910,148.464
C08003=1191.905,333.961,-73.590,-176.334,7.907,148.464
C08004=1191.909,333.713,-73.558,-176.337,7.903,148.463
C08005=1191.914,333.466,-73.526,-176.338,7.901,148.463
C08006=1191.917,333.218,-73.494,-176.341,7.898,148.463
C08007=1191.921,332.970,-73.462,-176.343,7.894,148.463
C08008=1191.925,332.721,-73.430,-176.346,7.891,148.463
C08009=1191.930,332.474,-73.398,-176.348,7.888,148.463
C08010=1191.933,332.226,-73.366,-176.350,7.885,148.463
C08011=1191.938,331.978,-73.334,-176.353,7.883,148.463
C08012=1191.942,331.730,-73.302,-176.355,7.879,148.462
C08013=1191.946,331.482,-73.270,-176.357,7.876,148.462
C08014=1191.951,331.235,-73.238,-176.360,7.873,148.462
C08015=1191.955,330.986,-73.207,-176.362,7.870,148.462
C08016=1191.958,330.738,-73.175,-176.364,7.867,148.462
C08017=1191.963,330.491,-73.143,-176.366,7.864,148.462
C08018=1191.967,330.243,-73.111,-176.369,7.861,148.462
C08019=1191.971,329.995,-73.079,-176.371,7.858,148.462
C08020=1191.975,329.747,-73.048,-176.374,7.854,148.461
C08021=1191.980,329.498,-73.016,-176.376,7.851,148.461
C08022=1191.984,329.251,-72.984,-176.378,7.849,148.461
C08023=1191.988,329.003,-72.952,-176.380,7.846,148.461
C08024=1191.992,328.755,-72.921,-176.383,7.843,148.461
C08025=1191.997,328.507,-72.889,-176.385,7.839,148.461
C08026=1192.001,328.259,-72.857,-176.388,7.836,148.461
C08027=1192.005,328.011,-72.826,-176.390,7.833,148.461
C08028=1192.009,327.763,-72.794,-176.392,7.831,148.461
C08029=1192.012,327.515,-72.762,-176.394,7.827,148.460
C08030=1192.018,327.267,-72.731,-176.397,7.824,148.460
C08031=1192.021,327.019,-72.699,-176.399,7.821,148.460
C08032=1192.026,326.772,-72.668,-176.402,7.818,148.460
C08033=1192.030,326.523,-72.636,-176.404,7.815,148.460
C08034=1192.034,326.276,-72.605,-176.406,7.813,148.460
C08035=1192.038,326.028,-72.573,-176.409,7.809,148.460
C08036=1192.042,325.779,-72.541,-176.411,7.806,148.460
C08037=1192.047,325.531,-72.510,-176.414,7.803,148.460
C08038=1192.051,325.283,-72.478,-176.416,7.800,148.460
C08039=1192.055,325.035,-72.447,-176.418,7.797,148.460
C08040=1192.059,324.787,-72.415,-176.421,7.794,148.460
C08041=1192.063,324.540,-72.384,-176.423,7.791,148.459
C08042=1192.067,324.291,-72.353,-176.426,7.788,148.459
C08043=1192.072,324.044,-72.321,-176.428,7.785,148.459
C08044=1192.076,323.795,-72.290,-176.431,7.782,148.459
C08045=1192.080,323.548,-72.259,-176.432,7.779,148.459
C08046=1192.084,323.299,-72.228,-176.435,7.776,148.459
C08047=1192.089,323.052,-72.196,-176.438,7.773,148.459
C08048=1192.093,322.804,-72.164,-176.440,7.770,148.459
C08049=1192.097,322.556,-72.133,-176.443,7.767,148.459
C08050=1192.101,322.308,-72.101,-176.444,7.764,148.459
C08051=1192.106,322.060,-72.070,-176.447,7.761,148.459
C08052=1192.110,321.811,-72.039,-176.449,7.758,148.458
C08053=1192.114,321.564,-72.008,-176.452,7.755,148.458
C08054=1192.118,321.315,-71.977,-176.455,7.752,148.458
C08055=1192.122,321.068,-71.945,-176.456,7.749,148.458
C08056=1192.126,320.819,-71.914,-176.459,7.746,148.458
C08057=1192.131,320.572,-71.882,-176.461,7.743,148.458
C08058=1192.134,320.324,-71.852,-176.464,7.740,148.458
C08059=1192.138,320.075,-71.821,-176.467,7.737,148.458
C08060=1192.143,319.828,-71.790,-176.468,7.735,148.458
C08061=1192.147,319.579,-71.759,-176.471,7.732,148.458
C08062=1192.151,319.331,-71.728,-176.474,7.729,148.458
C08063=1192.155,319.083,-71.696,-176.476,7.725,148.458
C08064=1192.160,318.835,-71.665,-176.479,7.722,148.458
C08065=1192.164,318.587,-71.634,-176.481,7.720,148.458
C08066=1192.168,318.339,-71.603,-176.483,7.717,148.458
C08067=1192.173,318.091,-71.572,-176.486,7.714,148.458
C08068=1192.177,317.843,-71.541,-176.488,7.710,148.457
C08069=1192.180,317.595,-71.511,-176.491,7.707,148.457
C08070=1192.185,317.348,-71.479,-176.493,7.705,148.457
C08071=1192.189,317.099,-71.448,-176.495,7.702,148.457
C08072=1192.193,316.851,-71.417,-176.498,7.699,148.457
C08073=1192.198,316.603,-71.386,-176.501,7.696,148.457
C08074=1192.202,316.355,-71.355,-176.503,7.693,148.457
C08075=1192.206,316.108,-71.324,-176.505,7.690,148.457
C08076=1192.210,315.859,-71.293,-176.508,7.687,148.457
C08077=1192.214,315.611,-71.262,-176.510,7.684,148.457
C08078=1192.219,315.363,-71.232,-176.513,7.681,148.457
C08079=1192.223,315.114,-71.201,-176.515,7.678,148.457
C08080=1192.228,314.838,-71.166,-176.518,7.675,148.457
C08081=1192.232,314.561,-71.132,-176.521,7.672,148.457
C08082=1192.237,314.286,-71.098,-176.523,7.669,148.457
C08083=1192.241,314.009,-71.063,-176.526,7.666,148.457
C08084=1192.246,313.761,-71.033,-176.528,7.663,148.457
C08085=1192.250,313.513,-71.002,-176.531,7.660,148.457
C08086=1192.255,313.265,-70.971,-176.533,7.656,148.457
C08087=1192.258,313.017,-70.941,-176.536,7.653,148.457
C08088=1192.263,312.769,-70.910,-176.538,7.651,148.457
C08089=1192.267,312.521,-70.879,-176.541,7.648,148.457
C08090=1192.271,312.273,-70.849,-176.543,7.645,148.456
C08091=1192.275,312.025,-70.818,-176.546,7.642,148.456
C08092=1192.280,311.777,-70.787,-176.548,7.640,148.456
C08093=1192.285,311.529,-70.756,-176.551,7.637,148.456
C08094=1192.288,311.280,-70.726,-176.553,7.633,148.456
C08095=1192.293,311.032,-70.696,-176.556,7.630,148.456
C08096=1192.297,310.784,-70.666,-176.558,7.627,148.456
C08097=1192.301,310.536,-70.635,-176.560,7.625,148.456
C08098=1192.305,310.288,-70.604,-176.563,7.622,148.456
C08099=1192.309,310.040,-70.573,-176.565,7.619,148.456
C08100=1192.314,309.792,-70.543,-176.568,7.616,148.456
C08101=1192.318,309.544,-70.512,-176.570,7.613,148.456
C08102=1192.322,309.295,-70.482,-176.573,7.610,148.456
C08103=1192.327,309.047,-70.451,-176.575,7.607,148.456
C08104=1192.330,308.799,-70.421,-176.578,7.604,148.456
C08105=1192.335,308.551,-70.390,-176.580,7.602,148.456
C08106=1192.340,308.303,-70.360,-176.583,7.599,148.456
C08107=1192.343,308.054,-70.330,-176.585,7.596,148.456
C08108=1192.348,307.807,-70.299,-176.588,7.593,148.456
C08109=1192.352,307.559,-70.269,-176.590,7.590,148.456
C08110=1192.357,307.310,-70.239,-176.592,7.587,148.456
C08111=1192.360,307.063,-70.209,-176.595,7.584,148.456
C08112=1192.365,306.815,-70.178,-176.598,7.581,148.456
C08113=1192.369,306.566,-70.148,-176.601,7.578,148.456
C08114=1192.373,306.318,-70.117,-176.602,7.576,148.456
C08115=1192.377,306.070,-70.087,-176.605,7.573,148.456
C08116=1192.382,305.822,-70.057,-176.608,7.570,148.456
C08117=1192.386,305.574,-70.027,-176.610,7.567,148.456
C08118=1192.391,305.326,-69.996,-176.612,7.565,148.456
C08119=1192.395,305.078,-69.967,-176.615,7.562,148.456
C08120=1192.399,304.829,-69.936,-176.617,7.558,148.456
C08121=1192.403,304.581,-69.906,-176.620,7.555,148.456
C08122=1192.408,304.333,-69.875,-176.622,7.553,148.456
C08123=1192.412,304.085,-69.846,-176.625,7.550,148.456
C08124=1192.416,303.837,-69.815,-176.628,7.547,148.456
C08125=1192.420,303.589,-69.785,-176.630,7.544,148.456
C08126=1192.424,303.341,-69.756,-176.633,7.542,148.456
C08127=1192.429,303.093,-69.725,-176.635,7.539,148.456
C08128=1192.433,302.844,-69.695,-176.637,7.536,148.456
C08129=1192.438,302.596,-69.665,-176.640,7.533,148.456
C08130=1192.442,302.348,-69.635,-176.642,7.530,148.456
C08131=1192.446,302.099,-69.605,-176.645,7.527,148.456
C08132=1192.450,301.851,-69.575,-176.648,7.524,148.456
C08133=1192.454,301.603,-69.545,-176.650,7.522,148.456
C08134=1192.458,301.355,-69.515,-176.653,7.519,148.456
C08135=1192.463,301.107,-69.485,-176.655,7.516,148.456
C08136=1192.467,300.859,-69.455,-176.658,7.513,148.456
C08137=1192.471,300.611,-69.425,-176.660,7.511,148.456
C08138=1192.476,300.362,-69.395,-176.662,7.508,148.456
C08139=1192.480,300.114,-69.366,-176.665,7.505,148.456
C08140=1192.484,299.866,-69.336,-176.668,7.502,148.456
C08141=1192.489,299.618,-69.305,-176.670,7.500,148.456
C08142=1192.493,299.370,-69.276,-176.673,7.496,148.456
C08143=1192.497,299.122,-69.246,-176.675,7.493,148.456
C08144=1192.501,298.874,-69.216,-176.678,7.491,148.456
C08145=1192.506,298.625,-69.186,-176.680,7.488,148.456
C08146=1192.510,298.377,-69.156,-176.683,7.485,148.456
C08147=1192.514,298.129,-69.127,-176.686,7.482,148.456
C08148=1192.519,297.881,-69.097,-176.688,7.480,148.456
C08149=1192.523,297.633,-69.068,-176.690,7.477,148.456
C08150=1192.528,297.384,-69.038,-176.693,7.474,148.456
C08151=1192.531,297.136,-69.008,-176.695,7.472,148.456
C08152=1192.536,296.888,-68.978,-176.698,7.469,148.456
C08153=1192.540,296.640,-68.949,-176.700,7.466,148.456
C08154=1192.544,296.392,-68.919,-176.703,7.463,148.456
C08155=1192.549,296.143,-68.889,-176.705,7.460,148.456
C08156=1192.553,295.895,-68.860,-176.708,7.457,148.456
C08157=1192.557,295.647,-68.830,-176.711,7.454,148.456
C08158=1192.561,295.399,-68.800,-176.713,7.452,148.456
C08159=1192.565,295.151,-68.771,-176.715,7.449,148.456
C08160=1192.570,294.902,-68.741,-176.718,7.446,148.456
C08161=1192.574,294.654,-68.712,-176.721,7.443,148.457
C08162=1192.578,294.406,-68.682,-176.723,7.441,148.457
C08163=1192.583,294.158,-68.653,-176.726,7.438,148.457
C08164=1192.588,293.910,-68.623,-176.728,7.435,148.457
C08165=1192.592,293.661,-68.594,-176.731,7.433,148.457
C08166=1192.596,293.413,-68.564,-176.733,7.430,148.457
C08167=1192.600,293.165,-68.535,-176.736,7.427,148.457
C08168=1192.604,292.917,-68.505,-176.738,7.425,148.457
C08169=1192.609,292.668,-68.476,-176.741,7.422,148.457
C08170=1192.613,292.420,-68.446,-176.744,7.419,148.457
C08171=1192.617,292.172,-68.417,-176.746,7.416,148.457
C08172=1192.621,291.923,-68.388,-176.748,7.413,148.457
C08173=1192.626,291.676,-68.358,-176.751,7.410,148.457
C08174=1192.630,291.428,-68.329,-176.754,7.407,148.457
C08175=1192.634,291.179,-68.300,-176.756,7.405,148.457
C08176=1192.639,290.930,-68.271,-176.759,7.402,148.457
C08177=1192.643,290.682,-68.241,-176.761,7.399,148.457
C08178=1192.647,290.434,-68.212,-176.763,7.397,148.457
C08179=1192.651,290.186,-68.182,-176.766,7.394,148.457
C08180=1192.656,289.938,-68.153,-176.769,7.391,148.457
C08181=1192.660,289.690,-68.124,-176.771,7.389,148.457
C08182=1192.665,289.441,-68.095,-176.774,7.386,148.457
C08183=1192.669,289.193,-68.066,-176.777,7.383,148.458
C08184=1192.673,288.919,-68.033,-176.780,7.380,148.458
C08185=1192.679,288.644,-68.001,-176.782,7.377,148.458
C08186=1192.683,288.369,-67.969,-176.785,7.374,148.458
C08187=1192.688,288.095,-67.937,-176.788,7.371,148.458
C08188=1192.692,287.847,-67.908,-176.790,7.369,148.458
C08189=1192.696,287.598,-67.879,-176.793,7.366,148.458
C08190=1192.700,287.350,-67.849,-176.795,7.363,148.458
C08191=1192.706,287.102,-67.821,-176.797,7.361,148.458
C08192=1192.710,286.854,-67.791,-176.800,7.358,148.458
C08193=1192.714,286.605,-67.762,-176.803,7.355,148.458
C08194=1192.718,286.357,-67.734,-176.806,7.353,148.458
C08195=1192.722,286.109,-67.705,-176.808,7.350,148.458
C08196=1192.727,285.861,-67.675,-176.811,7.347,148.458
C08197=1192.731,285.612,-67.646,-176.813,7.345,148.458
C08198=1192.735,285.364,-67.617,-176.816,7.342,148.458
C08199=1192.740,285.116,-67.589,-176.819,7.339,148.458
C08200=1192.744,284.868,-67.560,-176.821,7.337,148.459
C08201=1192.748,284.619,-67.530,-176.823,7.334,148.459
C08202=1192.753,284.371,-67.502,-176.826,7.331,148.459
C08203=1192.757,284.123,-67.472,-176.828,7.328,148.459
C08204=1192.761,283.874,-67.444,-176.831,7.325,148.459
C08205=1192.765,283.626,-67.415,-176.834,7.324,148.459
C08206=1192.770,283.378,-67.387,-176.836,7.321,148.459
C08207=1192.775,283.130,-67.357,-176.839,7.318,148.459
C08208=1192.778,282.881,-67.329,-176.841,7.315,148.459
C08209=1192.783,282.633,-67.300,-176.844,7.312,148.459
C08210=1192.788,282.385,-67.271,-176.847,7.309,148.459
C08211=1192.792,282.136,-67.242,-176.849,7.307,148.459
C08212=1192.796,281.888,-67.214,-176.851,7.304,148.459
C08213=1192.801,281.640,-67.185,-176.854,7.301,148.459
C08214=1192.805,281.391,-67.156,-176.857,7.299,148.460
C08215=1192.809,281.143,-67.128,-176.859,7.296,148.460
C08216=1192.814,280.894,-67.099,-176.862,7.294,148.460
C08217=1192.818,280.646,-67.070,-176.864,7.291,148.460
C08218=1192.822,280.398,-67.042,-176.867,7.288,148.460
C08219=1192.827,280.149,-67.013,-176.869,7.286,148.460
C08220=1192.831,279.901,-66.984,-176.872,7.283,148.460
C08221=1192.835,279.653,-66.956,-176.875,7.281,148.460
C08222=1192.840,279.404,-66.927,-176.877,7.278,148.460
C08223=1192.843,279.156,-66.898,-176.880,7.275,148.460
C08224=1192.848,278.908,-66.870,-176.882,7.273,148.460
C08225=1192.853,278.659,-66.841,-176.885,7.270,148.460
C08226=1192.857,278.412,-66.813,-176.888,7.267,148.460
C08227=1192.861,278.163,-66.784,-176.890,7.265,148.460
C08228=1192.865,277.915,-66.756,-176.893,7.262,148.461
C08229=1192.870,277.666,-66.728,-176.895,7.260,148.461
C08230=1192.874,277.418,-66.699,-176.898,7.257,148.461
C08231=1192.879,277.170,-66.671,-176.900,7.254,148.461
C08232=1192.883,276.921,-66.642,-176.903,7.252,148.461
C08233=1192.887,276.673,-66.613,-176.905,7.249,148.461
C08234=1192.892,276.425,-66.585,-176.908,7.247,148.461
C08235=1192.896,276.176,-66.557,-176.911,7.244,148.461
C08236=1192.901,275.928,-66.529,-176.913,7.242,148.461
C08237=1192.904,275.679,-66.500,-176.915,7.239,148.461
C08238=1192.910,275.431,-66.472,-176.918,7.236,148.461
C08239=1192.913,275.183,-66.443,-176.921,7.234,148.462
C08240=1192.918,274.935,-66.415,-176.924,7.231,148.462
C08241=1192.922,274.686,-66.387,-176.926,7.229,148.462
C08242=1192.926,274.439,-66.359,-176.928,7.226,148.462
C08243=1192.931,274.190,-66.330,-176.931,7.223,148.462
C08244=1192.934,273.941,-66.302,-176.933,7.221,148.462
C08245=1192.939,273.693,-66.274,-176.936,7.218,148.462
C08246=1192.943,273.444,-66.245,-176.939,7.216,148.462
C08247=1192.948,273.196,-66.217,-176.941,7.213,148.462
C08248=1192.952,272.948,-66.189,-176.943,7.210,148.463
C08249=1192.956,272.700,-66.161,-176.947,7.208,148.463
C08250=1192.961,272.451,-66.132,-176.949,7.205,148.463
C08251=1192.965,272.203,-66.105,-176.952,7.203,148.463
C08252=1192.970,271.953,-66.077,-176.954,7.200,148.463
C08253=1192.974,271.706,-66.049,-176.956,7.197,148.463
C08254=1192.979,271.458,-66.021,-176.960,7.195,148.463
C08255=1192.983,271.209,-65.992,-176.962,7.193,148.463
C08256=1192.988,270.961,-65.965,-176.964,7.190,148.463
C08257=1192.991,270.712,-65.936,-176.967,7.187,148.463
C08258=1192.996,270.464,-65.908,-176.970,7.185,148.464
C08259=1193.000,270.216,-65.880,-176.973,7.182,148.464
C08260=1193.005,269.967,-65.853,-176.975,7.180,148.464
C08261=1193.009,269.718,-65.824,-176.977,7.177,148.464
C08262=1193.014,269.470,-65.796,-176.980,7.174,148.464
C08263=1193.018,269.222,-65.769,-176.983,7.172,148.464
C08264=1193.022,268.974,-65.740,-176.985,7.170,148.464
C08265=1193.027,268.725,-65.713,-176.988,7.167,148.464
C08266=1193.031,268.476,-65.685,-176.990,7.164,148.464
C08267=1193.035,268.229,-65.657,-176.993,7.162,148.465
C08268=1193.040,267.980,-65.628,-176.995,7.160,148.465
C08269=1193.044,267.731,-65.601,-176.998,7.157,148.465
C08270=1193.049,267.483,-65.573,-177.000,7.154,148.465
C08271=1193.053,267.235,-65.545,-177.003,7.152,148.465
C08272=1193.057,266.986,-65.518,-177.006,7.149,148.465
C08273=1193.062,266.738,-65.490,-177.008,7.147,148.465
C08274=1193.066,266.490,-65.462,-177.011,7.144,148.466
C08275=1193.071,266.241,-65.434,-177.013,7.142,148.466
C08276=1193.075,265.993,-65.407,-177.016,7.139,148.466
C08277=1193.079,265.745,-65.379,-177.018,7.137,148.466
C08278=1193.084,265.496,-65.351,-177.021,7.134,148.466
C08279=1193.088,265.247,-65.323,-177.024,7.132,148.466
C08280=1193.093,264.999,-65.296,-177.026,7.129,148.466
C08281=1193.097,264.751,-65.268,-177.028,7.127,148.466
C08282=1193.101,264.502,-65.240,-177.032,7.124,148.467
C08283=1193.105,264.254,-65.213,-177.034,7.122,148.467
C08284=1193.111,264.005,-65.185,-177.036,7.119,148.467
C08285=1193.115,263.757,-65.157,-177.039,7.117,148.467
C08286=1193.119,263.508,-65.130,-177.042,7.114,148.467
C08287=1193.123,263.260,-65.102,-177.044,7.112,148.467
C08288=1193.128,262.987,-65.071,-177.047,7.109,148.467
C08289=1193.133,262.714,-65.042,-177.050,7.106,148.467
C08290=1193.138,262.442,-65.011,-177.053,7.103,148.468
C08291=1193.143,262.168,-64.981,-177.056,7.100,148.468
C08292=1193.147,261.920,-64.954,-177.058,7.098,148.468
C08293=1193.152,261.672,-64.926,-177.061,7.096,148.468
C08294=1193.156,261.423,-64.898,-177.063,7.093,148.468
C08295=1193.160,261.174,-64.871,-177.066,7.090,148.468
C08296=1193.165,260.926,-64.844,-177.069,7.089,148.468
C08297=1193.169,260.678,-64.817,-177.071,7.086,148.469
C08298=1193.173,260.429,-64.789,-177.074,7.083,148.469
C08299=1193.178,260.181,-64.761,-177.076,7.082,148.469
C08300=1193.182,259.932,-64.734,-177.079,7.079,148.469
C08301=1193.187,259.684,-64.707,-177.081,7.076,148.469
C08302=1193.191,259.435,-64.679,-177.084,7.074,148.469
C08303=1193.195,259.187,-64.652,-177.086,7.072,148.469
C08304=1193.200,258.938,-64.625,-177.089,7.069,148.469
C08305=1193.204,258.690,-64.597,-177.092,7.067,148.470
C08306=1193.209,258.442,-64.570,-177.094,7.064,148.470
C08307=1193.213,258.193,-64.543,-177.097,7.062,148.470
C08308=1193.217,257.945,-64.516,-177.100,7.059,148.470
C08309=1193.221,257.697,-64.488,-177.102,7.057,148.470
C08310=1193.226,257.448,-64.461,-177.105,7.054,148.470
C08311=1193.231,257.200,-64.434,-177.107,7.052,148.471
C08312=1193.235,256.951,-64.407,-177.110,7.049,148.471
C08313=1193.239,256.702,-64.380,-177.112,7.047,148.471
C08314=1193.244,256.454,-64.352,-177.115,7.045,148.471
C08315=1193.248,256.206,-64.325,-177.118,7.042,148.471
C08316=1193.253,255.957,-64.298,-177.120,7.040,148.471
C08317=1193.257,255.709,-64.271,-177.123,7.037,148.471
C08318=1193.261,255.460,-64.244,-177.125,7.035,148.472
C08319=1193.266,255.211,-64.217,-177.128,7.032,148.472
C08320=1193.270,254.963,-64.190,-177.130,7.030,148.472
C08321=1193.275,254.714,-64.163,-177.133,7.027,148.472
C08322=1193.280,254.466,-64.136,-177.136,7.025,148.472
C08323=1193.284,254.218,-64.109,-177.138,7.023,148.472
C08324=1193.288,253.969,-64.082,-177.141,7.020,148.473
C08325=1193.292,253.720,-64.055,-177.143,7.018,148.473
C08326=1193.297,253.471,-64.028,-177.146,7.015,148.473
C08327=1193.302,253.223,-64.001,-177.149,7.013,148.473
C08328=1193.306,252.975,-63.974,-177.151,7.010,148.473
C08329=1193.310,252.726,-63.947,-177.154,7.009,148.473
C08330=1193.315,252.478,-63.920,-177.156,7.006,148.474
C08331=1193.320,252.229,-63.893,-177.159,7.003,148.474
C08332=1193.323,251.981,-63.867,-177.161,7.002,148.474
C08333=1193.328,251.733,-63.840,-177.164,6.999,148.474
C08334=1193.333,251.484,-63.812,-177.167,6.997,148.474
C08335=1193.336,251.235,-63.786,-177.170,6.994,148.474
C08336=1193.341,250.987,-63.759,-177.172,6.992,148.474
C08337=1193.345,250.738,-63.731,-177.174,6.990,148.475
C08338=1193.350,250.490,-63.704,-177.177,6.987,148.475
C08339=1193.354,250.242,-63.678,-177.180,6.985,148.475
C08340=1193.359,249.992,-63.652,-177.182,6.982,148.475
C08341=1193.364,249.744,-63.625,-177.185,6.980,148.476
C08342=1193.368,249.496,-63.598,-177.187,6.978,148.476
C08343=1193.372,249.247,-63.571,-177.190,6.975,148.476
C08344=1193.376,248.999,-63.545,-177.193,6.973,148.476
C08345=1193.381,248.750,-63.518,-177.195,6.970,148.476
C08346=1193.386,248.501,-63.491,-177.198,6.968,148.476
C08347=1193.390,248.253,-63.465,-177.200,6.966,148.476
C08348=1193.394,248.005,-63.438,-177.203,6.963,148.477
C08349=1193.399,247.756,-63.411,-177.205,6.961,148.477
C08350=1193.403,247.507,-63.385,-177.209,6.959,148.477
C08351=1193.408,247.259,-63.358,-177.211,6.956,148.477
C08352=1193.412,247.011,-63.331,-177.213,6.954,148.477
C08353=1193.417,246.762,-63.305,-177.216,6.952,148.478
C08354=1193.421,246.513,-63.278,-177.218,6.949,148.478
C08355=1193.425,246.265,-63.251,-177.221,6.947,148.478
C08356=1193.430,246.016,-63.225,-177.224,6.945,148.478
C08357=1193.434,245.768,-63.199,-177.226,6.943,148.478
C08358=1193.439,245.519,-63.172,-177.229,6.940,148.478
C08359=1193.443,245.270,-63.146,-177.232,6.938,148.479
C08360=1193.448,245.022,-63.119,-177.234,6.936,148.479
C08361=1193.452,244.773,-63.093,-177.237,6.933,148.479
C08362=1193.457,244.525,-63.066,-177.239,6.931,148.479
C08363=1193.461,244.276,-63.039,-177.242,6.928,148.479
C08364=1193.465,244.027,-63.013,-177.245,6.926,148.480
C08365=1193.469,243.779,-62.987,-177.247,6.924,148.480
C08366=1193.475,243.531,-62.961,-177.250,6.921,148.480
C08367=1193.479,243.283,-62.934,-177.253,6.919,148.480
C08368=1193.483,243.034,-62.908,-177.255,6.917,148.480
C08369=1193.488,242.785,-62.881,-177.258,6.915,148.481
C08370=1193.492,242.536,-62.856,-177.260,6.912,148.481
C08371=1193.497,242.288,-62.829,-177.263,6.911,148.481
C08372=1193.501,242.039,-62.803,-177.265,6.908,148.481
C08373=1193.506,241.791,-62.776,-177.268,6.906,148.481
C08374=1193.510,241.542,-62.750,-177.270,6.904,148.482
C08375=1193.514,241.293,-62.724,-177.273,6.901,148.482
C08376=1193.519,241.045,-62.698,-177.276,6.899,148.482
C08377=1193.523,240.796,-62.672,-177.278,6.897,148.482
C08378=1193.528,240.548,-62.645,-177.281,6.894,148.482
C08379=1193.532,240.299,-62.619,-177.284,6.892,148.483
C08380=1193.537,240.050,-62.593,-177.286,6.889,148.483
C08381=1193.541,239.802,-62.566,-177.289,6.887,148.483
C08382=1193.545,239.553,-62.540,-177.291,6.885,148.483
C08383=1193.550,239.305,-62.515,-177.294,6.883,148.483
C08384=1193.555,239.056,-62.488,-177.296,6.880,148.483
C08385=1193.559,238.808,-62.462,-177.299,6.879,148.484
C08386=1193.563,238.559,-62.436,-177.301,6.876,148.484
C08387=1193.568,238.310,-62.409,-177.304,6.874,148.484
C08388=1193.572,238.061,-62.384,-177.307,6.872,148.485
C08389=1193.577,237.813,-62.358,-177.309,6.870,148.485
C08390=1193.581,237.565,-62.333,-177.312,6.867,148.485
C08391=1193.586,237.316,-62.305,-177.315,6.865,148.485
C08392=1193.591,237.044,-62.277,-177.318,6.862,148.485
C08393=1193.596,236.774,-62.249,-177.320,6.860,148.486
C08394=1193.600,236.502,-62.221,-177.323,6.857,148.486
C08395=1193.606,236.229,-62.192,-177.326,6.855,148.486
C08396=1193.610,235.981,-62.166,-177.329,6.853,148.486
C08397=1193.615,235.733,-62.141,-177.331,6.851,148.486
C08398=1193.619,235.484,-62.115,-177.334,6.848,148.487
C08399=1193.623,235.236,-62.089,-177.337,6.846,148.487
C08400=1193.628,234.986,-62.063,-177.339,6.844,148.487
C08401=1193.633,234.738,-62.037,-177.341,6.842,148.487
C08402=1193.637,234.490,-62.012,-177.345,6.839,148.487
C08403=1193.641,234.241,-61.985,-177.347,6.838,148.488
C08404=1193.645,233.993,-61.959,-177.349,6.835,148.488
C08405=1193.651,233.744,-61.933,-177.353,6.833,148.488
C08406=1193.655,233.495,-61.908,-177.355,6.831,148.488
C08407=1193.659,233.247,-61.882,-177.357,6.829,148.489
C08408=1193.663,232.998,-61.856,-177.360,6.827,148.489
C08409=1193.668,232.750,-61.831,-177.363,6.824,148.489
C08410=1193.672,232.501,-61.805,-177.365,6.822,148.489
C08411=1193.677,232.252,-61.779,-177.368,6.820,148.489
C08412=1193.681,232.004,-61.754,-177.371,6.817,148.490
C08413=1193.686,231.755,-61.727,-177.373,6.815,148.490
C08414=1193.691,231.506,-61.702,-177.376,6.813,148.490
C08415=1193.695,231.258,-61.676,-177.378,6.811,148.490
C08416=1193.700,231.009,-61.651,-177.381,6.808,148.491
C08417=1193.704,230.760,-61.625,-177.384,6.807,148.491
C08418=1193.708,230.511,-61.599,-177.386,6.804,148.491
C08419=1193.713,230.263,-61.574,-177.389,6.802,148.491
C08420=1193.718,230.014,-61.549,-177.392,6.800,148.492
C08421=1193.722,229.765,-61.523,-177.394,6.798,148.492
C08422=1193.727,229.517,-61.498,-177.396,6.796,148.492
C08423=1193.731,229.268,-61.472,-177.400,6.793,148.492
C08424=1193.736,229.020,-61.446,-177.402,6.791,148.492
C08425=1193.740,228.771,-61.421,-177.404,6.789,148.493
C08426=1193.744,228.522,-61.396,-177.407,6.787,148.493
C08427=1193.749,228.274,-61.370,-177.410,6.785,148.493
C08428=1193.753,228.025,-61.344,-177.412,6.783,148.493
C08429=1193.758,227.776,-61.319,-177.415,6.781,148.494
C08430=1193.762,227.528,-61.293,-177.417,6.779,148.494
C08431=1193.767,227.279,-61.268,-177.420,6.776,148.494
C08432=1193.772,227.031,-61.243,-177.423,6.774,148.494
C08433=1193.776,226.782,-61.217,-177.425,6.772,148.495
C08434=1193.780,226.533,-61.191,-177.428,6.769,148.495
C08435=1193.785,226.284,-61.167,-177.431,6.767,148.495
C08436=1193.790,226.035,-61.141,-177.433,6.766,148.495
C08437=1193.794,225.787,-61.116,-177.436,6.764,148.496
C08438=1193.798,225.538,-61.091,-177.438,6.762,148.496
C08439=1193.802,225.289,-61.065,-177.441,6.759,148.496
C08440=1193.807,225.041,-61.040,-177.444,6.757,148.496
C08441=1193.812,224.792,-61.015,-177.446,6.755,148.497
C08442=1193.817,224.544,-60.990,-177.449,6.753,148.497
C08443=1193.821,224.295,-60.964,-177.452,6.750,148.497
C08444=1193.826,224.046,-60.939,-177.454,6.748,148.497
C08445=1193.830,223.797,-60.913,-177.457,6.746,148.498
C08446=1193.835,223.549,-60.889,-177.459,6.745,148.498
C08447=1193.839,223.300,-60.864,-177.462,6.742,148.498
C08448=1193.843,223.051,-60.838,-177.465,6.740,148.498
C08449=1193.848,222.803,-60.813,-177.467,6.738,148.499
C08450=1193.852,222.554,-60.787,-177.470,6.736,148.499
C08451=1193.858,222.305,-60.763,-177.473,6.733,148.499
C08452=1193.861,222.057,-60.738,-177.476,6.731,148.499
C08453=1193.866,221.808,-60.713,-177.478,6.729,148.500
C08454=1193.870,221.559,-60.687,-177.480,6.727,148.500
C08455=1193.876,221.310,-60.663,-177.483,6.726,148.500
C08456=1193.879,221.062,-60.637,-177.486,6.723,148.500
C08457=1193.884,220.813,-60.613,-177.488,6.721,148.501
C08458=1193.888,220.564,-60.587,-177.491,6.719,148.501
C08459=1193.894,220.316,-60.562,-177.494,6.717,148.501
C08460=1193.897,220.067,-60.537,-177.496,6.714,148.501
C08461=1193.902,219.818,-60.512,-177.499,6.712,148.502
C08462=1193.907,219.570,-60.488,-177.502,6.711,148.502
C08463=1193.911,219.321,-60.462,-177.504,6.709,148.502
C08464=1193.916,219.073,-60.438,-177.506,6.707,148.502
C08465=1193.920,218.824,-60.412,-177.510,6.704,148.503
C08466=1193.925,218.575,-60.388,-177.512,6.702,148.503
C08467=1193.929,218.326,-60.363,-177.515,6.700,148.503
C08468=1193.934,218.078,-60.338,-177.517,6.698,148.504
C08469=1193.938,217.828,-60.313,-177.520,6.696,148.504
C08470=1193.943,217.580,-60.289,-177.523,6.694,148.504
C08471=1193.948,217.332,-60.263,-177.525,6.691,148.504
C08472=1193.952,217.082,-60.238,-177.528,6.690,148.505
C08473=1193.957,216.834,-60.214,-177.530,6.688,148.505
C08474=1193.961,216.585,-60.189,-177.533,6.686,148.505
C08475=1193.965,216.337,-60.164,-177.536,6.683,148.505
C08476=1193.970,216.087,-60.139,-177.539,6.681,148.506
C08477=1193.975,215.839,-60.115,-177.541,6.679,148.506
C08478=1193.979,215.590,-60.091,-177.544,6.678,148.506
C08479=1193.983,215.341,-60.065,-177.546,6.675,148.506
C08480=1193.988,215.093,-60.041,-177.549,6.673,148.507
C08481=1193.993,214.844,-60.016,-177.552,6.671,148.507
C08482=1193.997,214.595,-59.991,-177.555,6.669,148.507
C08483=1194.002,214.346,-59.967,-177.557,6.667,148.508
C08484=1194.006,214.097,-59.942,-177.559,6.665,148.508
C08485=1194.011,213.849,-59.917,-177.562,6.663,148.508
C08486=1194.016,213.601,-59.892,-177.565,6.661,148.509
C08487=1194.019,213.351,-59.868,-177.567,6.659,148.509
C08488=1194.025,213.103,-59.843,-177.570,6.657,148.509
C08489=1194.029,212.854,-59.819,-177.573,6.655,148.509
C08490=1194.033,212.605,-59.794,-177.575,6.653,148.510
C08491=1194.038,212.356,-59.770,-177.579,6.650,148.510
C08492=1194.043,212.108,-59.745,-177.581,6.648,148.510
C08493=1194.047,211.859,-59.721,-177.583,6.647,148.510
C08494=1194.052,211.610,-59.696,-177.586,6.645,148.511
C08495=1194.056,211.361,-59.672,-177.589,6.643,148.511
C08496=1194.061,211.091,-59.646,-177.592,6.640,148.511
C08497=1194.066,210.820,-59.618,-177.595,6.638,148.512
C08498=1194.071,210.550,-59.592,-177.597,6.636,148.512
C08499=1194.076,210.280,-59.565,-177.600,6.634,148.512
C08500=1194.081,210.031,-59.542,-177.603,6.632,148.513
C08501=1194.086,209.782,-59.517,-177.605,6.630,148.513
C08502=1194.090,209.533,-59.493,-177.608,6.628,148.513
C08503=1194.094,209.285,-59.468,-177.611,6.626,148.513
C08504=1194.099,209.035,-59.443,-177.613,6.623,148.514
C08505=1194.103,208.787,-59.419,-177.616,6.622,148.514
C08506=1194.108,208.538,-59.395,-177.619,6.620,148.514
C08507=1194.113,208.290,-59.371,-177.621,6.618,148.515
C08508=1194.117,208.041,-59.346,-177.624,6.616,148.515
C08509=1194.122,207.792,-59.322,-177.626,6.614,148.515
C08510=1194.126,207.543,-59.298,-177.629,6.611,148.515
C08511=1194.131,207.295,-59.274,-177.632,6.610,148.516
C08512=1194.136,207.046,-59.249,-177.635,6.608,148.516
C08513=1194.140,206.797,-59.225,-177.637,6.606,148.516
C08514=1194.144,206.548,-59.201,-177.640,6.604,148.517
C08515=1194.149,206.300,-59.176,-177.642,6.602,148.517
C08516=1194.154,206.051,-59.153,-177.645,6.600,148.517
C08517=1194.158,205.802,-59.129,-177.647,6.598,148.518
C08518=1194.163,205.553,-59.104,-177.651,6.596,148.518
C08519=1194.167,205.304,-59.080,-177.653,6.594,148.518
C08520=1194.172,205.055,-59.056,-177.655,6.592,148.518
C08521=1194.176,204.807,-59.032,-177.658,6.590,148.519
C08522=1194.182,204.558,-59.008,-177.661,6.588,148.519
C08523=1194.186,204.308,-58.984,-177.663,6.586,148.519
C08524=1194.190,204.060,-58.960,-177.666,6.584,148.520
C08525=1194.194,203.812,-58.936,-177.669,6.583,148.520
C08526=1194.200,203.563,-58.911,-177.671,6.581,148.520
C08527=1194.204,203.314,-58.888,-177.674,6.578,148.520
C08528=1194.209,203.065,-58.864,-177.677,6.576,148.521
C08529=1194.213,202.816,-58.840,-177.679,6.574,148.521
C08530=1194.217,202.567,-58.816,-177.682,6.572,148.522
C08531=1194.222,202.319,-58.791,-177.685,6.571,148.522
C08532=1194.227,202.069,-58.768,-177.687,6.568,148.522
C08533=1194.231,201.821,-58.744,-177.690,6.567,148.522
C08534=1194.236,201.572,-58.720,-177.692,6.565,148.523
C08535=1194.240,201.324,-58.696,-177.695,6.563,148.523
C08536=1194.245,201.075,-58.672,-177.698,6.560,148.523
C08537=1194.250,200.825,-58.648,-177.701,6.559,148.524
C08538=1194.254,200.577,-58.624,-177.703,6.557,148.524
C08539=1194.259,200.328,-58.600,-177.706,6.555,148.524
C08540=1194.263,200.079,-58.576,-177.708,6.553,148.524
C08541=1194.268,199.830,-58.553,-177.711,6.551,148.525
C08542=1194.272,199.582,-58.529,-177.714,6.549,148.525
C08543=1194.277,199.333,-58.506,-177.716,6.547,148.526
C08544=1194.281,199.084,-58.482,-177.719,6.546,148.526
C08545=1194.286,198.835,-58.458,-177.722,6.544,148.526
C08546=1194.291,198.587,-58.433,-177.724,6.542,148.527
C08547=1194.296,198.338,-58.410,-177.726,6.540,148.527
C08548=1194.301,198.089,-58.387,-177.729,6.538,148.527
C08549=1194.304,197.839,-58.362,-177.732,6.535,148.527
C08550=1194.309,197.590,-58.339,-177.735,6.534,148.528
C08551=1194.313,197.342,-58.315,-177.738,6.532,148.528
C08552=1194.318,197.093,-58.292,-177.740,6.530,148.528
C08553=1194.323,196.844,-58.268,-177.743,6.528,148.529
C08554=1194.327,196.596,-58.244,-177.746,6.526,148.529
C08555=1194.332,196.347,-58.221,-177.748,6.524,148.529
C08556=1194.337,196.097,-58.197,-177.750,6.522,148.530
C08557=1194.341,195.849,-58.173,-177.753,6.521,148.530
C08558=1194.346,195.600,-58.150,-177.756,6.519,148.530
C08559=1194.350,195.351,-58.127,-177.758,6.517,148.531
C08560=1194.355,195.103,-58.103,-177.761,6.515,148.531
C08561=1194.360,194.854,-58.079,-177.764,6.513,148.531
C08562=1194.364,194.605,-58.056,-177.766,6.512,148.532
C08563=1194.369,194.356,-58.032,-177.769,6.510,148.532
C08564=1194.373,194.107,-58.008,-177.772,6.508,148.532
C08565=1194.378,193.858,-57.985,-177.774,6.506,148.532
C08566=1194.383,193.609,-57.962,-177.777,6.503,148.533
C08567=1194.387,193.360,-57.939,-177.780,6.501,148.533
C08568=1194.391,193.111,-57.916,-177.782,6.500,148.533
C08569=1194.396,192.863,-57.891,-177.785,6.498,148.534
C08570=1194.401,192.615,-57.868,-177.788,6.496,148.534
C08571=1194.406,192.366,-57.845,-177.790,6.494,148.535
C08572=1194.411,192.116,-57.822,-177.793,6.492,148.535
C08573=1194.415,191.867,-57.798,-177.796,6.491,148.535
C08574=1194.420,191.618,-57.775,-177.798,6.489,148.536
C08575=1194.425,191.369,-57.752,-177.801,6.487,148.536
C08576=1194.428,191.121,-57.728,-177.804,6.485,148.536
C08577=1194.433,190.872,-57.705,-177.806,6.483,148.536
C08578=1194.438,190.623,-57.681,-177.808,6.481,148.537
C08579=1194.442,190.374,-57.658,-177.811,6.479,148.537
C08580=1194.447,190.125,-57.635,-177.814,6.478,148.537
C08581=1194.452,189.876,-57.611,-177.816,6.476,148.538
C08582=1194.456,189.627,-57.589,-177.819,6.474,148.538
C08583=1194.461,189.379,-57.566,-177.822,6.472,148.539
C08584=1194.466,189.130,-57.542,-177.824,6.470,148.539
C08585=1194.470,188.881,-57.519,-177.827,6.469,148.539
C08586=1194.475,188.632,-57.496,-177.830,6.467,148.540
C08587=1194.479,188.383,-57.473,-177.832,6.465,148.540
C08588=1194.484,188.134,-57.449,-177.835,6.463,148.540
C08589=1194.488,187.885,-57.426,-177.838,6.461,148.541
C08590=1194.493,187.636,-57.403,-177.840,6.460,148.541
C08591=1194.498,187.388,-57.380,-177.843,6.458,148.541
C08592=1194.502,187.139,-57.357,-177.846,6.456,148.542
C08593=1194.507,186.890,-57.334,-177.848,6.454,148.542
C08594=1194.512,186.641,-57.310,-177.851,6.452,148.542
C08595=1194.516,186.392,-57.287,-177.853,6.450,148.543
C08596=1194.521,186.143,-57.265,-177.856,6.448,148.543
C08597=1194.526,185.894,-57.242,-177.859,6.447,148.543
C08598=1194.530,185.646,-57.219,-177.861,6.445,148.544
C08599=1194.535,185.397,-57.196,-177.864,6.443,148.544
C08600=1194.540,185.127,-57.171,-177.867,6.441,148.544
C08601=1194.545,184.857,-57.146,-177.870,6.440,148.545
C08602=1194.550,184.588,-57.121,-177.873,6.437,148.545
C08603=1194.555,184.318,-57.096,-177.876,6.435,148.546
C08604=1194.559,184.069,-57.073,-177.878,6.434,148.546
C08605=1194.564,183.820,-57.050,-177.881,6.432,148.546
C08606=1194.569,183.572,-57.028,-177.884,6.430,148.547
C08607=1194.574,183.322,-57.005,-177.886,6.428,148.547
C08608=1194.578,183.073,-56.982,-177.889,6.426,148.547
C08609=1194.582,182.825,-56.959,-177.892,6.425,148.548
C08610=1194.587,182.576,-56.936,-177.894,6.423,148.548
C08611=1194.592,182.327,-56.914,-177.897,6.421,148.548
C08612=1194.596,182.078,-56.890,-177.900,6.419,148.549
C08613=1194.601,181.829,-56.867,-177.902,6.417,148.549
C08614=1194.605,181.580,-56.844,-177.905,6.416,148.549
C08615=1194.611,181.331,-56.822,-177.907,6.415,148.550
C08616=1194.615,181.083,-56.799,-177.910,6.413,148.550
C08617=1194.620,180.833,-56.777,-177.912,6.411,148.551
C08618=1194.624,180.584,-56.754,-177.915,6.409,148.551
C08619=1194.629,180.336,-56.731,-177.918,6.407,148.551
C08620=1194.633,180.086,-56.709,-177.920,6.406,148.552
C08621=1194.638,179.837,-56.686,-177.923,6.404,148.552
C08622=1194.643,179.589,-56.663,-177.926,6.402,148.552
C08623=1194.648,179.340,-56.640,-177.928,6.400,148.553
C08624=1194.651,179.091,-56.618,-177.931,6.398,148.553
C08625=1194.656,178.841,-56.595,-177.934,6.397,148.553
C08626=1194.661,178.593,-56.573,-177.936,6.395,148.554
C08627=1194.666,178.344,-56.550,-177.939,6.393,148.554
C08628=1194.670,178.095,-56.527,-177.942,6.391,148.555
C08629=1194.676,177.846,-56.505,-177.944,6.389,148.555
C08630=1194.680,177.597,-56.482,-177.947,6.388,148.555
C08631=1194.685,177.348,-56.460,-177.950,6.386,148.556
C08632=1194.689,177.100,-56.437,-177.952,6.384,148.556
C08633=1194.694,176.850,-56.415,-177.954,6.383,148.556
C08634=1194.698,176.601,-56.392,-177.957,6.381,148.557
C08635=1194.703,176.353,-56.370,-177.960,6.379,148.557
C08636=1194.708,176.104,-56.347,-177.962,6.378,148.557
C08637=1194.712,175.854,-56.325,-177.965,6.376,148.558
C08638=1194.717,175.606,-56.302,-177.968,6.374,148.558
C08639=1194.722,175.357,-56.280,-177.970,6.372,148.559
C08640=1194.726,175.108,-56.258,-177.973,6.370,148.559
C08641=1194.731,174.859,-56.235,-177.976,6.369,148.559
C08642=1194.735,174.610,-56.213,-177.978,6.367,148.560
C08643=1194.740,174.362,-56.190,-177.981,6.365,148.560
C08644=1194.745,174.112,-56.168,-177.984,6.363,148.560
C08645=1194.749,173.863,-56.145,-177.986,6.362,148.561
C08646=1194.754,173.614,-56.122,-177.989,6.361,148.561
C08647=1194.759,173.365,-56.100,-177.991,6.359,148.561
C08648=1194.764,173.116,-56.079,-177.994,6.357,148.562
C08649=1194.768,172.868,-56.056,-177.997,6.355,148.562
C08650=1194.773,172.619,-56.034,-177.999,6.353,148.563
C08651=1194.777,172.369,-56.012,-178.002,6.352,148.563
C08652=1194.782,172.120,-55.990,-178.005,6.350,148.563
C08653=1194.787,171.872,-55.967,-178.008,6.348,148.564
C08654=1194.791,171.622,-55.945,-178.010,6.347,148.564
C08655=1194.796,171.374,-55.923,-178.013,6.346,148.565
C08656=1194.801,171.124,-55.900,-178.015,6.344,148.565
C08657=1194.806,170.876,-55.878,-178.018,6.342,148.565
C08658=1194.810,170.627,-55.856,-178.021,6.340,148.566
C08659=1194.815,170.378,-55.834,-178.023,6.338,148.566
C08660=1194.820,170.128,-55.811,-178.026,6.337,148.566
C08661=1194.824,169.879,-55.789,-178.029,6.335,148.567
C08662=1194.829,169.631,-55.767,-178.031,6.333,148.567
C08663=1194.833,169.382,-55.745,-178.034,6.331,148.567
C08664=1194.838,169.133,-55.723,-178.036,6.330,148.568
C08665=1194.843,168.883,-55.701,-178.039,6.328,148.568
C08666=1194.848,168.635,-55.679,-178.042,6.327,148.569
C08667=1194.852,168.385,-55.657,-178.045,6.325,148.569
C08668=1194.857,168.137,-55.635,-178.047,6.323,148.570
C08669=1194.861,167.887,-55.613,-178.050,6.322,148.570
C08670=1194.867,167.638,-55.591,-178.053,6.320,148.570
C08671=1194.871,167.390,-55.568,-178.055,6.319,148.571
C08672=1194.876,167.141,-55.546,-178.057,6.317,148.571
C08673=1194.880,166.892,-55.524,-178.060,6.315,148.571
C08674=1194.885,166.643,-55.503,-178.063,6.314,148.572
C08675=1194.890,166.394,-55.481,-178.065,6.312,148.572
C08676=1194.894,166.145,-55.459,-178.068,6.310,148.573
C08677=1194.899,165.896,-55.437,-178.071,6.308,148.573
C08678=1194.904,165.647,-55.415,-178.073,6.308,148.574
C08679=1194.909,165.398,-55.393,-178.076,6.306,148.574
C08680=1194.913,165.149,-55.371,-178.079,6.304,148.574
C08681=1194.918,164.900,-55.349,-178.081,6.302,148.575
C08682=1194.922,164.651,-55.327,-178.084,6.300,148.575
C08683=1194.927,164.402,-55.306,-178.087,6.299,148.575
C08684=1194.931,164.152,-55.284,-178.089,6.297,148.576
C08685=1194.936,163.904,-55.263,-178.091,6.296,148.576
C08686=1194.941,163.655,-55.241,-178.094,6.294,148.576
C08687=1194.945,163.406,-55.219,-178.097,6.293,148.577
C08688=1194.950,163.157,-55.197,-178.100,6.291,148.577
C08689=1194.955,162.908,-55.175,-178.103,6.289,148.578
C08690=1194.959,162.659,-55.153,-178.105,6.287,148.578
C08691=1194.964,162.410,-55.132,-178.107,6.286,148.579
C08692=1194.969,162.161,-55.110,-178.110,6.285,148.579
C08693=1194.974,161.912,-55.089,-178.113,6.283,148.579
C08694=1194.978,161.662,-55.067,-178.115,6.281,148.580
C08695=1194.983,161.414,-55.045,-178.119,6.279,148.580
C08696=1194.988,161.165,-55.023,-178.121,6.278,148.581
C08697=1194.992,160.916,-55.001,-178.123,6.277,148.581
C08698=1194.997,160.666,-54.980,-178.126,6.275,148.581
C08699=1195.002,160.418,-54.959,-178.129,6.273,148.582
C08700=1195.006,160.168,-54.937,-178.131,6.271,148.582
C08701=1195.011,159.920,-54.915,-178.134,6.270,148.583
C08702=1195.016,159.671,-54.894,-178.136,6.269,148.583
C08703=1195.021,159.421,-54.872,-178.139,6.267,148.584
C08704=1195.025,159.152,-54.849,-178.142,6.265,148.584
C08705=1195.031,158.883,-54.825,-178.145,6.264,148.584
C08706=1195.035,158.614,-54.802,-178.148,6.262,148.585
C08707=1195.041,158.345,-54.779,-178.151,6.260,148.585
C08708=1195.046,158.096,-54.757,-178.153,6.259,148.586
C08709=1195.051,157.848,-54.735,-178.156,6.257,148.586
C08710=1195.054,157.598,-54.715,-178.159,6.255,148.586
C08711=1195.059,157.349,-54.693,-178.161,6.253,148.587
C08712=1195.064,157.101,-54.671,-178.164,6.253,148.587
C08713=1195.069,156.852,-54.650,-178.166,6.251,148.588
C08714=1195.074,156.602,-54.628,-178.169,6.249,148.588
C08715=1195.079,156.353,-54.607,-178.172,6.247,148.588
C08716=1195.083,156.105,-54.586,-178.175,6.246,148.589
C08717=1195.087,155.855,-54.564,-178.177,6.245,148.589
C08718=1195.092,155.606,-54.543,-178.180,6.243,148.590
C08719=1195.097,155.357,-54.522,-178.182,6.241,148.590
C08720=1195.102,155.108,-54.501,-178.185,6.240,148.591
C08721=1195.107,154.859,-54.479,-178.187,6.239,148.591
C08722=1195.111,154.610,-54.458,-178.190,6.237,148.591
C08723=1195.116,154.361,-54.437,-178.193,6.235,148.592
C08724=1195.121,154.112,-54.416,-178.196,6.234,148.592
C08725=1195.125,153.863,-54.394,-178.198,6.232,148.593
C08726=1195.130,153.614,-54.373,-178.201,6.231,148.593
C08727=1195.135,153.365,-54.351,-178.203,6.229,148.593
C08728=1195.140,153.116,-54.331,-178.206,6.227,148.594
C08729=1195.145,152.867,-54.309,-178.209,6.226,148.594
C08730=1195.149,152.617,-54.288,-178.211,6.225,148.595
C08731=1195.154,152.368,-54.267,-178.214,6.223,148.595
C08732=1195.159,152.120,-54.245,-178.217,6.221,148.596
C08733=1195.164,151.870,-54.224,-178.219,6.220,148.596
C08734=1195.167,151.621,-54.203,-178.221,6.219,148.596
C08735=1195.172,151.372,-54.182,-178.225,6.217,148.597
C08736=1195.178,151.123,-54.161,-178.227,6.215,148.597
C08737=1195.182,150.874,-54.140,-178.230,6.214,148.598
C08738=1195.187,150.625,-54.119,-178.232,6.213,148.598
C08739=1195.192,150.377,-54.097,-178.235,6.211,148.598
C08740=1195.196,150.127,-54.077,-178.238,6.209,148.599
C08741=1195.201,149.878,-54.056,-178.241,6.208,148.599
C08742=1195.206,149.628,-54.035,-178.243,6.207,148.600
C08743=1195.210,149.380,-54.014,-178.245,6.205,148.600
C08744=1195.215,149.131,-53.993,-178.248,6.203,148.601
C08745=1195.221,148.882,-53.972,-178.251,6.202,148.601
C08746=1195.224,148.632,-53.950,-178.253,6.201,148.602
C08747=1195.229,148.383,-53.929,-178.256,6.199,148.602
C08748=1195.234,148.134,-53.909,-178.259,6.197,148.602
C08749=1195.239,147.885,-53.888,-178.261,6.195,148.603
C08750=1195.244,147.636,-53.866,-178.264,6.195,148.603
C08751=1195.248,147.387,-53.846,-178.267,6.193,148.604
C08752=1195.253,147.138,-53.825,-178.269,6.191,148.604
C08753=1195.258,146.889,-53.805,-178.272,6.190,148.604
C08754=1195.262,146.639,-53.783,-178.275,6.189,148.605
C08755=1195.266,146.391,-53.762,-178.277,6.187,148.605
C08756=1195.272,146.142,-53.741,-178.280,6.185,148.606
C08757=1195.276,145.893,-53.721,-178.282,6.184,148.606
C08758=1195.281,145.643,-53.700,-178.285,6.183,148.607
C08759=1195.286,145.394,-53.679,-178.288,6.181,148.607
C08760=1195.291,145.145,-53.658,-178.291,6.179,148.608
C08761=1195.296,144.897,-53.637,-178.293,6.178,148.608
C08762=1195.300,144.648,-53.616,-178.295,6.177,148.608
C08763=1195.305,144.398,-53.595,-178.299,6.175,148.609
C08764=1195.310,144.149,-53.575,-178.301,6.174,148.609
C08765=1195.314,143.901,-53.555,-178.303,6.173,148.610
C08766=1195.319,143.651,-53.533,-178.306,6.171,148.610
C08767=1195.323,143.402,-53.513,-178.309,6.169,148.611
C08768=1195.328,143.152,-53.492,-178.311,6.168,148.611
C08769=1195.333,142.903,-53.472,-178.314,6.167,148.612
C08770=1195.338,142.654,-53.451,-178.317,6.165,148.612
C08771=1195.342,142.405,-53.430,-178.319,6.164,148.613
C08772=1195.348,142.156,-53.409,-178.322,6.162,148.613
C08773=1195.352,141.907,-53.389,-178.325,6.161,148.613
C08774=1195.356,141.658,-53.369,-178.327,6.160,148.614
C08775=1195.362,141.409,-53.348,-178.330,6.158,148.614
C08776=1195.366,141.160,-53.327,-178.333,6.157,148.615
C08777=1195.371,140.911,-53.306,-178.335,6.155,148.615
C08778=1195.376,140.662,-53.286,-178.337,6.154,148.616
C08779=1195.380,140.413,-53.266,-178.341,6.152,148.616
C08780=1195.385,140.163,-53.245,-178.343,6.151,148.617
C08781=1195.390,139.914,-53.224,-178.345,6.150,148.617
C08782=1195.395,139.665,-53.203,-178.348,6.148,148.617
C08783=1195.399,139.416,-53.183,-178.351,6.146,148.618
C08784=1195.404,139.167,-53.163,-178.353,6.146,148.618
C08785=1195.409,138.917,-53.142,-178.356,6.144,148.619
C08786=1195.414,138.668,-53.122,-178.359,6.142,148.619
C08787=1195.418,138.420,-53.102,-178.361,6.141,148.620
C08788=1195.423,138.170,-53.081,-178.364,6.140,148.620
C08789=1195.428,137.921,-53.060,-178.367,6.138,148.620
C08790=1195.433,137.672,-53.041,-178.369,6.137,148.621
C08791=1195.437,137.423,-53.020,-178.372,6.135,148.621
C08792=1195.442,137.174,-52.999,-178.375,6.134,148.622
C08793=1195.447,136.925,-52.979,-178.377,6.133,148.622
C08794=1195.452,136.676,-52.959,-178.380,6.131,148.623
C08795=1195.457,136.426,-52.939,-178.383,6.130,148.623
C08796=1195.462,136.178,-52.918,-178.385,6.129,148.624
C08797=1195.466,135.929,-52.898,-178.388,6.127,148.624
C08798=1195.470,135.680,-52.877,-178.391,6.125,148.625
C08799=1195.476,135.430,-52.857,-178.393,6.124,148.625
C08800=1195.480,135.181,-52.837,-178.395,6.123,148.625
C08801=1195.485,134.932,-52.816,-178.399,6.121,148.626
C08802=1195.489,134.683,-52.796,-178.401,6.120,148.626
C08803=1195.495,134.433,-52.776,-178.403,6.119,148.627
C08804=1195.500,134.185,-52.756,-178.407,6.117,148.627
C08805=1195.504,133.936,-52.735,-178.409,6.116,148.628
C08806=1195.509,133.686,-52.716,-178.411,6.114,148.628
C08807=1195.513,133.437,-52.695,-178.414,6.113,148.629
C08808=1195.519,133.168,-52.674,-178.417,6.112,148.629
C08809=1195.524,132.900,-52.652,-178.419,6.110,148.630
C08810=1195.529,132.631,-52.630,-178.423,6.109,148.630
C08811=1195.535,132.363,-52.608,-178.425,6.107,148.631
C08812=1195.539,132.113,-52.588,-178.428,6.107,148.631
C08813=1195.544,131.864,-52.568,-178.431,6.105,148.632
C08814=1195.549,131.615,-52.548,-178.433,6.103,148.632
C08815=1195.553,131.366,-52.528,-178.436,6.102,148.633
C08816=1195.558,131.116,-52.508,-178.439,6.101,148.633
C08817=1195.563,130.868,-52.488,-178.441,6.099,148.633
C08818=1195.568,130.618,-52.468,-178.444,6.098,148.634
C08819=1195.573,130.369,-52.447,-178.447,6.096,148.635
C08820=1195.577,130.120,-52.428,-178.449,6.096,148.635
C08821=1195.582,129.871,-52.407,-178.452,6.094,148.636
C08822=1195.587,129.622,-52.388,-178.455,6.092,148.636
C08823=1195.592,129.373,-52.368,-178.457,6.091,148.636
C08824=1195.596,129.123,-52.348,-178.460,6.090,148.637
C08825=1195.601,128.874,-52.328,-178.462,6.088,148.637
C08826=1195.606,128.625,-52.308,-178.465,6.087,148.638
C08827=1195.611,128.377,-52.288,-178.468,6.086,148.638
C08828=1195.615,128.127,-52.268,-178.470,6.085,148.639
C08829=1195.620,127.878,-52.248,-178.473,6.083,148.639
C08830=1195.624,127.629,-52.228,-178.476,6.082,148.640
C08831=1195.629,127.379,-52.209,-178.478,6.081,148.640
C08832=1195.634,127.131,-52.189,-178.481,6.079,148.641
C08833=1195.639,126.881,-52.169,-178.483,6.078,148.641
C08834=1195.643,126.632,-52.149,-178.486,6.077,148.642
C08835=1195.648,126.383,-52.129,-178.489,6.075,148.642
C08836=1195.654,126.134,-52.110,-178.491,6.074,148.643
C08837=1195.658,125.885,-52.089,-178.494,6.073,148.643
C08838=1195.663,125.635,-52.070,-178.496,6.072,148.643
C08839=1195.667,125.386,-52.050,-178.499,6.070,148.644
C08840=1195.673,125.137,-52.030,-178.501,6.069,148.644
C08841=1195.677,124.888,-52.010,-178.504,6.068,148.645
C08842=1195.682,124.638,-51.991,-178.507,6.066,148.645
C08843=1195.687,124.390,-51.971,-178.509,6.065,148.646
C08844=1195.692,124.141,-51.951,-178.512,6.063,148.646
C08845=1195.697,123.891,-51.931,-178.515,6.063,148.647
C08846=1195.701,123.641,-51.912,-178.517,6.061,148.647
C08847=1195.706,123.393,-51.892,-178.520,6.059,148.648
C08848=1195.711,123.144,-51.872,-178.523,6.059,148.648
C08849=1195.715,122.894,-51.853,-178.525,6.057,148.649
C08850=1195.720,122.645,-51.834,-178.528,6.056,148.649
C08851=1195.725,122.396,-51.814,-178.531,6.055,148.650
C08852=1195.730,122.147,-51.794,-178.533,6.054,148.650
C08853=1195.735,121.898,-51.774,-178.536,6.052,148.651
C08854=1195.740,121.648,-51.755,-178.539,6.050,148.651
C08855=1195.744,121.399,-51.735,-178.541,6.050,148.652
C08856=1195.750,121.150,-51.716,-178.544,6.048,148.652
C08857=1195.754,120.901,-51.697,-178.546,6.047,148.653
C08858=1195.758,120.652,-51.676,-178.549,6.046,148.653
C08859=1195.764,120.403,-51.657,-178.551,6.045,148.654
C08860=1195.768,120.153,-51.638,-178.554,6.043,148.654
C08861=1195.773,119.904,-51.618,-178.557,6.042,148.655
C08862=1195.778,119.655,-51.599,-178.559,6.041,148.655
C08863=1195.782,119.406,-51.579,-178.562,6.039,148.655
C08864=1195.787,119.156,-51.560,-178.565,6.038,148.656
C08865=1195.792,118.907,-51.541,-178.567,6.037,148.657
C08866=1195.797,118.658,-51.521,-178.570,6.036,148.657
C08867=1195.803,118.409,-51.502,-178.573,6.034,148.658
C08868=1195.807,118.160,-51.483,-178.575,6.033,148.658
C08869=1195.811,117.910,-51.463,-178.578,6.032,148.659
C08870=1195.817,117.661,-51.444,-178.580,6.031,148.659
C08871=1195.821,117.412,-51.424,-178.583,6.030,148.660
C08872=1195.826,117.163,-51.405,-178.585,6.029,148.660
C08873=1195.831,116.913,-51.386,-178.588,6.027,148.660
C08874=1195.835,116.664,-51.366,-178.591,6.026,148.661
C08875=1195.841,116.415,-51.347,-178.593,6.025,148.661
C08876=1195.845,116.166,-51.328,-178.597,6.023,148.662
C08877=1195.850,115.917,-51.308,-178.599,6.022,148.663
C08878=1195.855,115.667,-51.289,-178.601,6.020,148.663
C08879=1195.860,115.419,-51.270,-178.604,6.020,148.664
C08880=1195.864,115.169,-51.250,-178.607,6.018,148.664
C08881=1195.870,114.920,-51.231,-178.609,6.018,148.665
C08882=1195.874,114.671,-51.212,-178.612,6.016,148.665
C08883=1195.878,114.422,-51.192,-178.614,6.015,148.665
C08884=1195.884,114.173,-51.173,-178.617,6.013,148.666
C08885=1195.888,113.923,-51.155,-178.619,6.013,148.666
C08886=1195.893,113.674,-51.135,-178.623,6.011,148.667
C08887=1195.898,113.424,-51.116,-178.625,6.010,148.667
C08888=1195.903,113.176,-51.097,-178.627,6.008,148.668
C08889=1195.907,112.926,-51.077,-178.630,6.008,148.669
C08890=1195.913,112.677,-51.058,-178.633,6.006,148.669
C08891=1195.917,112.427,-51.040,-178.635,6.006,148.670
C08892=1195.922,112.179,-51.020,-178.638,6.004,148.670
C08893=1195.926,111.929,-51.001,-178.641,6.003,148.671
C08894=1195.932,111.680,-50.982,-178.643,6.001,148.671
C08895=1195.937,111.431,-50.962,-178.646,6.000,148.671
C08896=1195.941,111.182,-50.944,-178.649,5.999,148.672
C08897=1195.946,110.932,-50.925,-178.651,5.998,148.672
C08898=1195.951,110.684,-50.906,-178.654,5.997,148.673
C08899=1195.956,110.434,-50.886,-178.656,5.996,148.674
C08900=1195.960,110.185,-50.868,-178.659,5.994,148.674
C08901=1195.965,109.935,-50.849,-178.661,5.994,148.675
C08902=1195.971,109.686,-50.829,-178.664,5.992,148.675
C08903=1195.975,109.437,-50.812,-178.667,5.991,148.676
C08904=1195.980,109.188,-50.792,-178.669,5.989,148.676
C08905=1195.985,108.939,-50.773,-178.672,5.989,148.677
C08906=1195.990,108.689,-50.754,-178.675,5.987,148.677
C08907=1195.994,108.440,-50.736,-178.677,5.987,148.678
C08908=1195.999,108.191,-50.716,-178.680,5.985,148.678
C08909=1196.004,107.942,-50.698,-178.683,5.984,148.679
C08910=1196.009,107.692,-50.678,-178.685,5.982,148.679
C08911=1196.013,107.444,-50.660,-178.688,5.982,148.680
C08912=1196.019,107.175,-50.640,-178.691,5.980,148.680
C08913=1196.023,106.907,-50.619,-178.693,5.980,148.681
C08914=1196.029,106.638,-50.599,-178.696,5.978,148.681
C08915=1196.035,106.369,-50.579,-178.699,5.976,148.682
C08916=1196.039,106.120,-50.560,-178.701,5.975,148.682
C08917=1196.044,105.871,-50.541,-178.705,5.974,148.683
C08918=1196.049,105.621,-50.522,-178.707,5.973,148.683
C08919=1196.053,105.373,-50.504,-178.710,5.972,148.684
C08920=1196.059,105.123,-50.485,-178.712,5.971,148.684
C08921=1196.063,104.874,-50.466,-178.715,5.970,148.685
C08922=1196.069,104.625,-50.447,-178.717,5.968,148.685
C08923=1196.073,104.376,-50.429,-178.720,5.968,148.686
C08924=1196.078,104.126,-50.410,-178.723,5.966,148.686
C08925=1196.083,103.877,-50.391,-178.725,5.966,148.687
C08926=1196.087,103.628,-50.373,-178.728,5.964,148.688
C08927=1196.093,103.379,-50.353,-178.731,5.963,148.688
C08928=1196.097,103.129,-50.335,-178.733,5.962,148.689
C08929=1196.102,102.880,-50.317,-178.735,5.961,148.689
C08930=1196.107,102.631,-50.298,-178.739,5.959,148.690
C08931=1196.112,102.382,-50.280,-178.741,5.958,148.690
C08932=1196.116,102.132,-50.261,-178.743,5.958,148.691
C08933=1196.122,101.883,-50.242,-178.746,5.956,148.691
C08934=1196.127,101.634,-50.224,-178.749,5.955,148.692
C08935=1196.131,101.384,-50.205,-178.751,5.954,148.692
C08936=1196.136,101.135,-50.187,-178.754,5.953,148.693
C08937=1196.141,100.886,-50.168,-178.757,5.951,148.693
C08938=1196.146,100.637,-50.150,-178.759,5.951,148.694
C08939=1196.151,100.387,-50.131,-178.761,5.950,148.694
C08940=1196.155,100.138,-50.112,-178.765,5.948,148.695
C08941=1196.160,99.889,-50.094,-178.767,5.947,148.695
C08942=1196.165,99.639,-50.076,-178.770,5.946,148.696
C08943=1196.170,99.391,-50.057,-178.772,5.945,148.696
C08944=1196.175,99.141,-50.039,-178.775,5.944,148.697
C08945=1196.179,98.891,-50.020,-178.777,5.943,148.697
C08946=1196.184,98.642,-50.002,-178.780,5.942,148.698
C08947=1196.189,98.393,-49.983,-178.783,5.941,148.698
C08948=1196.194,98.144,-49.965,-178.785,5.940,148.699
C08949=1196.199,97.894,-49.947,-178.788,5.938,148.700
C08950=1196.204,97.645,-49.929,-178.791,5.938,148.700
C08951=1196.209,97.396,-49.909,-178.793,5.936,148.701
C08952=1196.214,97.147,-49.892,-178.796,5.935,148.701
C08953=1196.218,96.897,-49.873,-178.798,5.934,148.702
C08954=1196.223,96.648,-49.855,-178.801,5.933,148.702
C08955=1196.228,96.399,-49.837,-178.803,5.932,148.703
C08956=1196.233,96.150,-49.818,-178.807,5.931,148.703
C08957=1196.238,95.901,-49.800,-178.809,5.930,148.704
C08958=1196.243,95.651,-49.782,-178.811,5.929,148.704
C08959=1196.247,95.402,-49.764,-178.814,5.928,148.705
C08960=1196.252,95.153,-49.746,-178.817,5.927,148.706
C08961=1196.257,94.903,-49.728,-178.819,5.925,148.706
C08962=1196.262,94.653,-49.709,-178.822,5.925,148.707
C08963=1196.267,94.405,-49.690,-178.824,5.924,148.707
C08964=1196.272,94.156,-49.672,-178.827,5.922,148.708
C08965=1196.277,93.906,-49.654,-178.830,5.921,148.708
C08966=1196.282,93.657,-49.636,-178.833,5.920,148.709
C08967=1196.287,93.408,-49.618,-178.835,5.919,148.709
C08968=1196.291,93.158,-49.600,-178.837,5.919,148.710
C08969=1196.296,92.909,-49.582,-178.840,5.917,148.710
C08970=1196.301,92.660,-49.564,-178.843,5.916,148.711
C08971=1196.306,92.410,-49.545,-178.845,5.915,148.711
C08972=1196.311,92.161,-49.527,-178.848,5.914,148.712
C08973=1196.316,91.911,-49.509,-178.851,5.913,148.713
C08974=1196.321,91.662,-49.491,-178.853,5.912,148.713
C08975=1196.325,91.413,-49.473,-178.856,5.911,148.714
C08976=1196.330,91.164,-49.455,-178.858,5.910,148.714
C08977=1196.335,90.915,-49.437,-178.861,5.909,148.715
C08978=1196.340,90.665,-49.419,-178.864,5.908,148.715
C08979=1196.345,90.416,-49.401,-178.866,5.907,148.716
C08980=1196.349,90.166,-49.383,-178.869,5.906,148.716
C08981=1196.354,89.917,-49.365,-178.872,5.905,148.717
C08982=1196.359,89.668,-49.347,-178.874,5.903,148.717
C08983=1196.364,89.419,-49.329,-178.877,5.903,148.718
C08984=1196.369,89.170,-49.311,-178.879,5.902,148.718
C08985=1196.374,88.920,-49.293,-178.882,5.900,148.719
C08986=1196.379,88.671,-49.275,-178.884,5.899,148.719
C08987=1196.384,88.421,-49.258,-178.887,5.899,148.720
C08988=1196.389,88.172,-49.240,-178.890,5.897,148.721
C08989=1196.394,87.923,-49.222,-178.892,5.897,148.721
C08990=1196.398,87.673,-49.203,-178.895,5.896,148.722
C08991=1196.403,87.424,-49.185,-178.898,5.894,148.722
C08992=1196.408,87.175,-49.167,-178.900,5.894,148.723
C08993=1196.413,86.926,-49.149,-178.903,5.892,148.723
C08994=1196.418,86.676,-49.132,-178.906,5.891,148.724
C08995=1196.423,86.427,-49.114,-178.908,5.891,148.724
C08996=1196.428,86.178,-49.096,-178.911,5.889,148.725
C08997=1196.432,85.929,-49.079,-178.913,5.888,148.725
C08998=1196.437,85.680,-49.061,-178.916,5.888,148.726
C08999=1196.442,85.430,-49.043,-178.919,5.886,148.727
C09000=1196.447,85.181,-49.025,-178.921,5.885,148.727
C09001=1196.452,84.931,-49.007,-178.924,5.885,148.728
C09002=1196.457,84.682,-48.989,-178.926,5.883,148.728
C09003=1196.462,84.432,-48.972,-178.929,5.882,148.729
C09004=1196.467,84.183,-48.954,-178.931,5.882,148.729
C09005=1196.471,83.934,-48.937,-178.934,5.880,148.730
C09006=1196.476,83.685,-48.919,-178.937,5.880,148.731
C09007=1196.481,83.435,-48.902,-178.939,5.879,148.731
C09008=1196.486,83.186,-48.884,-178.942,5.877,148.732
C09009=1196.491,82.937,-48.866,-178.944,5.876,148.732
C09010=1196.497,82.687,-48.848,-178.947,5.876,148.733
C09011=1196.501,82.438,-48.830,-178.950,5.874,148.733
C09012=1196.506,82.189,-48.813,-178.952,5.874,148.734
C09013=1196.511,81.939,-48.796,-178.955,5.873,148.734
C09014=1196.516,81.690,-48.778,-178.958,5.871,148.735
C09015=1196.521,81.440,-48.761,-178.960,5.871,148.735
C09016=1196.526,81.172,-48.741,-178.962,5.870,148.736
C09017=1196.531,80.903,-48.722,-178.966,5.868,148.737
C09018=1196.536,80.635,-48.704,-178.968,5.868,148.737
C09019=1196.541,80.366,-48.685,-178.971,5.867,148.738
C09020=1196.547,80.118,-48.667,-178.974,5.866,148.738
C09021=1196.552,79.869,-48.649,-178.976,5.865,148.739
C09022=1196.557,79.619,-48.632,-178.979,5.864,148.740
C09023=1196.561,79.370,-48.615,-178.982,5.863,148.740
C09024=1196.566,79.120,-48.597,-178.984,5.862,148.741
C09025=1196.571,78.871,-48.579,-178.987,5.860,148.741
C09026=1196.576,78.622,-48.563,-178.990,5.860,148.742
C09027=1196.581,78.373,-48.545,-178.992,5.859,148.742
C09028=1196.586,78.123,-48.527,-178.995,5.858,148.743
C09029=1196.591,77.874,-48.510,-178.998,5.857,148.743
C09030=1196.595,77.624,-48.493,-179.000,5.856,148.744
C09031=1196.600,77.375,-48.475,-179.002,5.856,148.745
C09032=1196.605,77.125,-48.458,-179.005,5.854,148.745
C09033=1196.609,76.876,-48.440,-179.008,5.853,148.746
C09034=1196.615,76.627,-48.423,-179.010,5.853,148.746
C09035=1196.620,76.378,-48.405,-179.013,5.851,148.747
C09036=1196.625,76.129,-48.389,-179.016,5.851,148.747
C09037=1196.630,75.879,-48.371,-179.018,5.850,148.748
C09038=1196.635,75.630,-48.353,-179.020,5.849,148.748
C09039=1196.639,75.380,-48.337,-179.024,5.848,148.749
C09040=1196.644,75.131,-48.319,-179.026,5.847,148.750
C09041=1196.649,74.881,-48.302,-179.028,5.846,148.750
C09042=1196.654,74.632,-48.285,-179.031,5.845,148.751
C09043=1196.659,74.383,-48.267,-179.034,5.844,148.751
C09044=1196.664,74.134,-48.251,-179.036,5.843,148.752
C09045=1196.669,73.884,-48.233,-179.038,5.842,148.752
C09046=1196.674,73.635,-48.215,-179.042,5.841,148.753
C09047=1196.678,73.385,-48.199,-179.044,5.840,148.753
C09048=1196.684,73.135,-48.181,-179.046,5.840,148.754
C09049=1196.688,72.887,-48.164,-179.049,5.839,148.755
C09050=1196.694,72.637,-48.147,-179.052,5.837,148.755
C09051=1196.699,72.388,-48.130,-179.054,5.837,148.756
C09052=1196.703,72.139,-48.112,-179.057,5.836,148.756
C09053=1196.708,71.889,-48.095,-179.059,5.835,148.757
C09054=1196.713,71.639,-48.079,-179.062,5.834,148.758
C09055=1196.719,71.390,-48.062,-179.065,5.833,148.758
C09056=1196.723,71.142,-48.044,-179.067,5.833,148.759
C09057=1196.728,70.892,-48.027,-179.070,5.831,148.759
C09058=1196.732,70.642,-48.010,-179.073,5.830,148.760
C09059=1196.738,70.392,-47.993,-179.075,5.830,148.760
C09060=1196.743,70.144,-47.977,-179.077,5.829,148.761
C09061=1196.748,69.895,-47.959,-179.081,5.827,148.762
C09062=1196.752,69.645,-47.942,-179.083,5.827,148.762
C09063=1196.757,69.395,-47.925,-179.085,5.826,148.763
C09064=1196.762,69.146,-47.908,-179.088,5.825,148.763
C09065=1196.768,68.897,-47.891,-179.091,5.824,148.764
C09066=1196.772,68.648,-47.874,-179.093,5.823,148.764
C09067=1196.777,68.398,-47.857,-179.096,5.823,148.765
C09068=1196.782,68.149,-47.840,-179.098,5.822,148.765
C09069=1196.787,67.899,-47.823,-179.101,5.821,148.766
C09070=1196.792,67.650,-47.806,-179.104,5.820,148.767
C09071=1196.797,67.400,-47.789,-179.106,5.819,148.767
C09072=1196.802,67.151,-47.772,-179.109,5.818,148.768
C09073=1196.807,66.902,-47.756,-179.111,5.818,148.769
C09074=1196.812,66.652,-47.739,-179.114,5.816,148.769
C09075=1196.816,66.403,-47.721,-179.117,5.816,148.770
C09076=1196.821,66.153,-47.704,-179.119,5.815,148.770
C09077=1196.826,65.905,-47.688,-179.121,5.814,148.771
C09078=1196.831,65.655,-47.671,-179.125,5.813,148.771
C09079=1196.836,65.405,-47.654,-179.127,5.812,148.772
C09080=1196.840,65.156,-47.637,-179.129,5.811,148.773
C09081=1196.846,64.907,-47.620,-179.132,5.811,148.773
C09082=1196.851,64.657,-47.604,-179.134,5.810,148.774
C09083=1196.855,64.408,-47.587,-179.137,5.809,148.774
C09084=1196.861,64.159,-47.570,-179.140,5.808,148.775
C09085=1196.866,63.909,-47.554,-179.142,5.807,148.775
C09086=1196.870,63.660,-47.537,-179.145,5.807,148.776
C09087=1196.876,63.411,-47.520,-179.148,5.805,148.777
C09088=1196.880,63.161,-47.503,-179.150,5.804,148.777
C09089=1196.885,62.912,-47.487,-179.153,5.804,148.778
C09090=1196.891,62.663,-47.470,-179.155,5.803,148.778
C09091=1196.895,62.412,-47.454,-179.158,5.802,148.779
C09092=1196.900,62.163,-47.437,-179.161,5.801,148.780
C09093=1196.906,61.914,-47.420,-179.163,5.800,148.780
C09094=1196.910,61.664,-47.404,-179.166,5.799,148.781
C09095=1196.915,61.415,-47.387,-179.168,5.799,148.781
C09096=1196.920,61.166,-47.371,-179.171,5.798,148.782
C09097=1196.925,60.916,-47.353,-179.174,5.797,148.782
C09098=1196.929,60.667,-47.337,-179.176,5.796,148.783
C09099=1196.935,60.418,-47.320,-179.178,5.795,148.783
C09100=1196.939,60.168,-47.304,-179.181,5.795,148.784
C09101=1196.945,59.918,-47.287,-179.184,5.794,148.785
C09102=1196.950,59.669,-47.271,-179.186,5.792,148.785
C09103=1196.954,59.420,-47.254,-179.189,5.792,148.786
C09104=1196.959,59.171,-47.238,-179.192,5.791,148.787
C09105=1196.965,58.921,-47.221,-179.194,5.790,148.787
C09106=1196.969,58.671,-47.205,-179.196,5.790,148.788
C09107=1196.974,58.422,-47.188,-179.199,5.789,148.788
C09108=1196.979,58.173,-47.172,-179.202,5.788,148.789
C09109=1196.985,57.924,-47.155,-179.204,5.787,148.789
C09110=1196.989,57.674,-47.139,-179.207,5.787,148.790
C09111=1196.994,57.424,-47.122,-179.209,5.786,148.791
C09112=1196.999,57.176,-47.106,-179.212,5.785,148.791
C09113=1197.003,56.926,-47.089,-179.215,5.784,148.792
C09114=1197.010,56.676,-47.073,-179.218,5.783,148.793
C09115=1197.014,56.427,-47.056,-179.220,5.782,148.793
C09116=1197.019,56.178,-47.040,-179.222,5.782,148.794
C09117=1197.024,55.928,-47.024,-179.225,5.781,148.794
C09118=1197.028,55.678,-47.007,-179.227,5.780,148.795
C09119=1197.033,55.430,-46.991,-179.230,5.779,148.795
C09120=1197.038,55.160,-46.974,-179.233,5.779,148.796
C09121=1197.044,54.892,-46.955,-179.236,5.778,148.797
C09122=1197.050,54.624,-46.938,-179.239,5.777,148.797
C09123=1197.055,54.355,-46.920,-179.241,5.776,148.798
C09124=1197.060,54.106,-46.905,-179.244,5.775,148.799
C09125=1197.064,53.856,-46.888,-179.246,5.775,148.799
C09126=1197.070,53.607,-46.872,-179.248,5.774,148.800
C09127=1197.074,53.358,-46.856,-179.252,5.772,148.800
C09128=1197.080,53.108,-46.839,-179.254,5.772,148.801
C09129=1197.085,52.858,-46.823,-179.257,5.771,148.802
C09130=1197.090,52.610,-46.807,-179.259,5.770,148.802
C09131=1197.095,52.359,-46.791,-179.262,5.770,148.803
C09132=1197.100,52.111,-46.774,-179.264,5.769,148.803
C09133=1197.104,51.861,-46.758,-179.266,5.769,148.804
C09134=1197.110,51.612,-46.742,-179.270,5.767,148.805
C09135=1197.114,51.362,-46.725,-179.272,5.767,148.805
C09136=1197.120,51.113,-46.710,-179.275,5.766,148.806
C09137=1197.124,50.863,-46.693,-179.277,5.765,148.806
C09138=1197.129,50.614,-46.678,-179.280,5.765,148.807
C09139=1197.134,50.365,-46.661,-179.282,5.764,148.807
C09140=1197.139,50.115,-46.645,-179.285,5.763,148.808
C09141=1197.144,49.866,-46.629,-179.288,5.762,148.809
